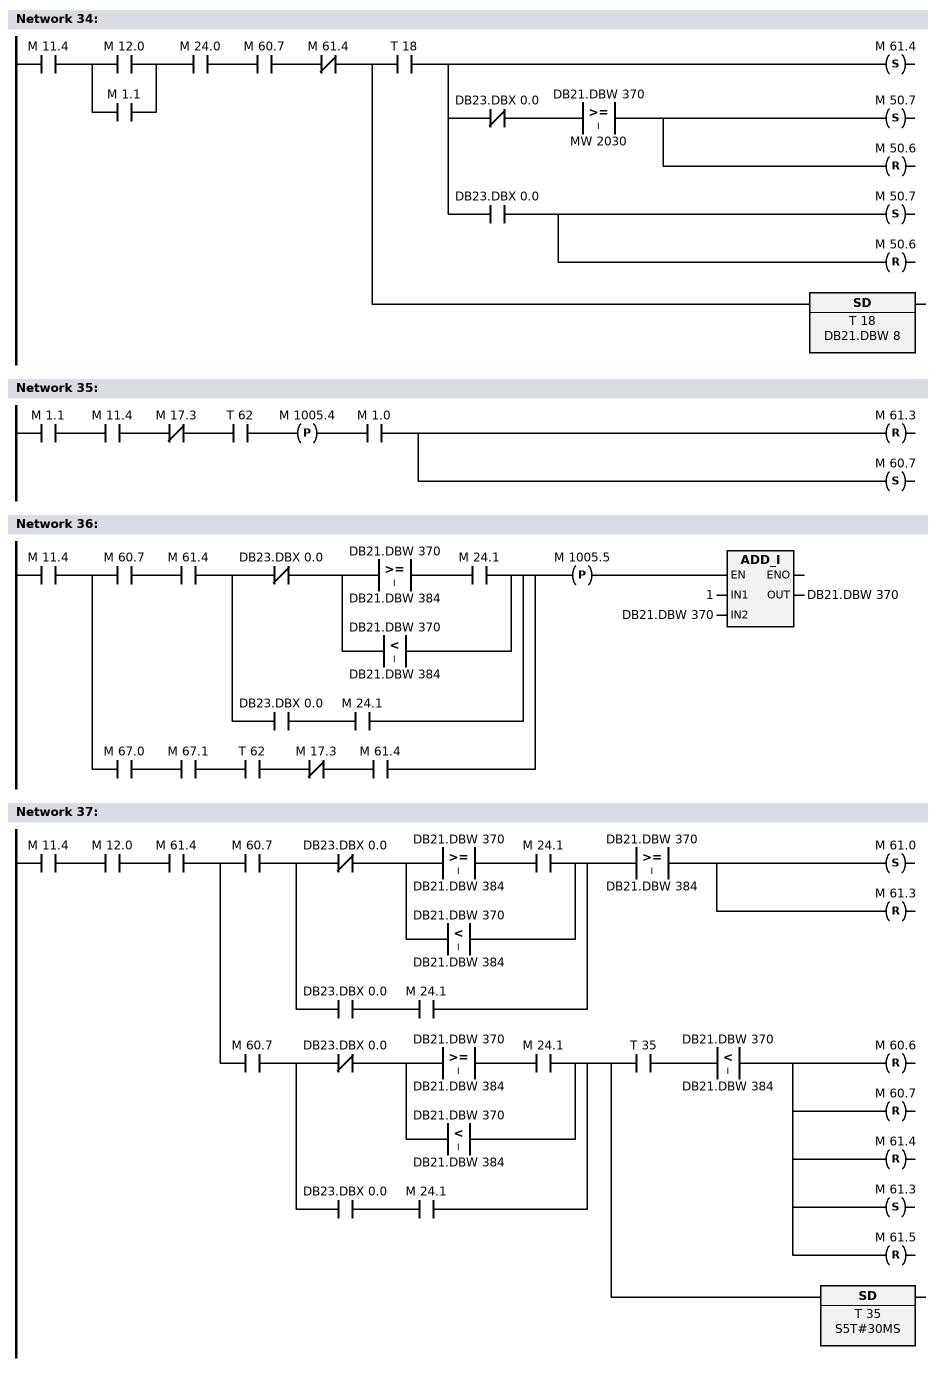
NETWORK
TITLE =
      A     M 11.4;
      A(;
      O     M 12.0;
      O     M 1.1;
      );
      A     M 24.0;
      A     M 60.7;
      AN    M 61.4;
      =     L 24.0;
      A     L 24.0;
      A     T 18;
      =     L 24.1;
      A     L 24.1;
      BLD   102;
      S     M 61.4;
      A     L 24.1;
      AN    DB23.DBX 0.0;
      A(;
      L     DB21.DBW 370;
      L     MW 2030;
      >=I;
      );
      S     M 50.7;
      R     M 50.6;
      A     L 24.1;
      A     DB23.DBX 0.0;
      S     M 50.7;
      R     M 50.6;
      A     L 24.0;
      BLD   102;
      L     DB21.DBW 8;
      SD    T 18;
NETWORK
TITLE =
      A     M 1.1;
      A     M 11.4;
      AN    M 17.3;
      A     T 62;
      FP    M 1005.4;
      A     M 1.0;
      R     M 61.3;
      S     M 60.7;
NETWORK
TITLE =
      A     M 11.4;
      A(;
      A     M 60.7;
      A     M 61.4;
      A(;
      AN    DB23.DBX 0.0;
      A(;
      A(;
      L     DB21.DBW 370;
      L     DB21.DBW 384;
      >=I;
      );
      A     M 24.1;
      O(;
      L     DB21.DBW 370;
      L     DB21.DBW 384;
      <I;
      );
      );
      O;
      A     DB23.DBX 0.0;
      A     M 24.1;
      );
      O;
      A     M 67.0;
      A     M 67.1;
      A     T 62;
      AN    M 17.3;
      A     M 61.4;
      );
      FP    M 1005.5;
      JNB   M025;
      L     1;
      L     DB21.DBW 370;
      +I;
      T     DB21.DBW 370;
M025: NOP   0;
NETWORK
TITLE =
      A     M 11.4;
      A     M 12.0;
      A     M 61.4;
      =     L 24.0;
      A     L 24.0;
      A     M 60.7;
      A(;
      AN    DB23.DBX 0.0;
      A(;
      A(;
      L     DB21.DBW 370;
      L     DB21.DBW 384;
      >=I;
      );
      A     M 24.1;
      O(;
      L     DB21.DBW 370;
      L     DB21.DBW 384;
      <I;
      );
      );
      O;
      A     DB23.DBX 0.0;
      A     M 24.1;
      );
      A(;
      L     DB21.DBW 370;
      L     DB21.DBW 384;
      >=I;
      );
      S     M 61.0;
      R     M 61.3;
      A     L 24.0;
      A     M 60.7;
      A(;
      AN    DB23.DBX 0.0;
      A(;
      A(;
      L     DB21.DBW 370;
      L     DB21.DBW 384;
      >=I;
      );
      A     M 24.1;
      O(;
      L     DB21.DBW 370;
      L     DB21.DBW 384;
      <I;
      );
      );
      O;
      A     DB23.DBX 0.0;
      A     M 24.1;
      );
      =     L 24.1;
      A     L 24.1;
      A     T 35;
      A(;
      L     DB21.DBW 370;
      L     DB21.DBW 384;
      <I;
      );
      R     M 60.6;
      R     M 60.7;
      R     M 61.4;
      S     M 61.3;
      R     M 61.5;
      A     L 24.1;
      BLD   102;
      L     S5T#30MS;
      SD    T 35;
NETWORK
TITLE =
NETWORK
TITLE =
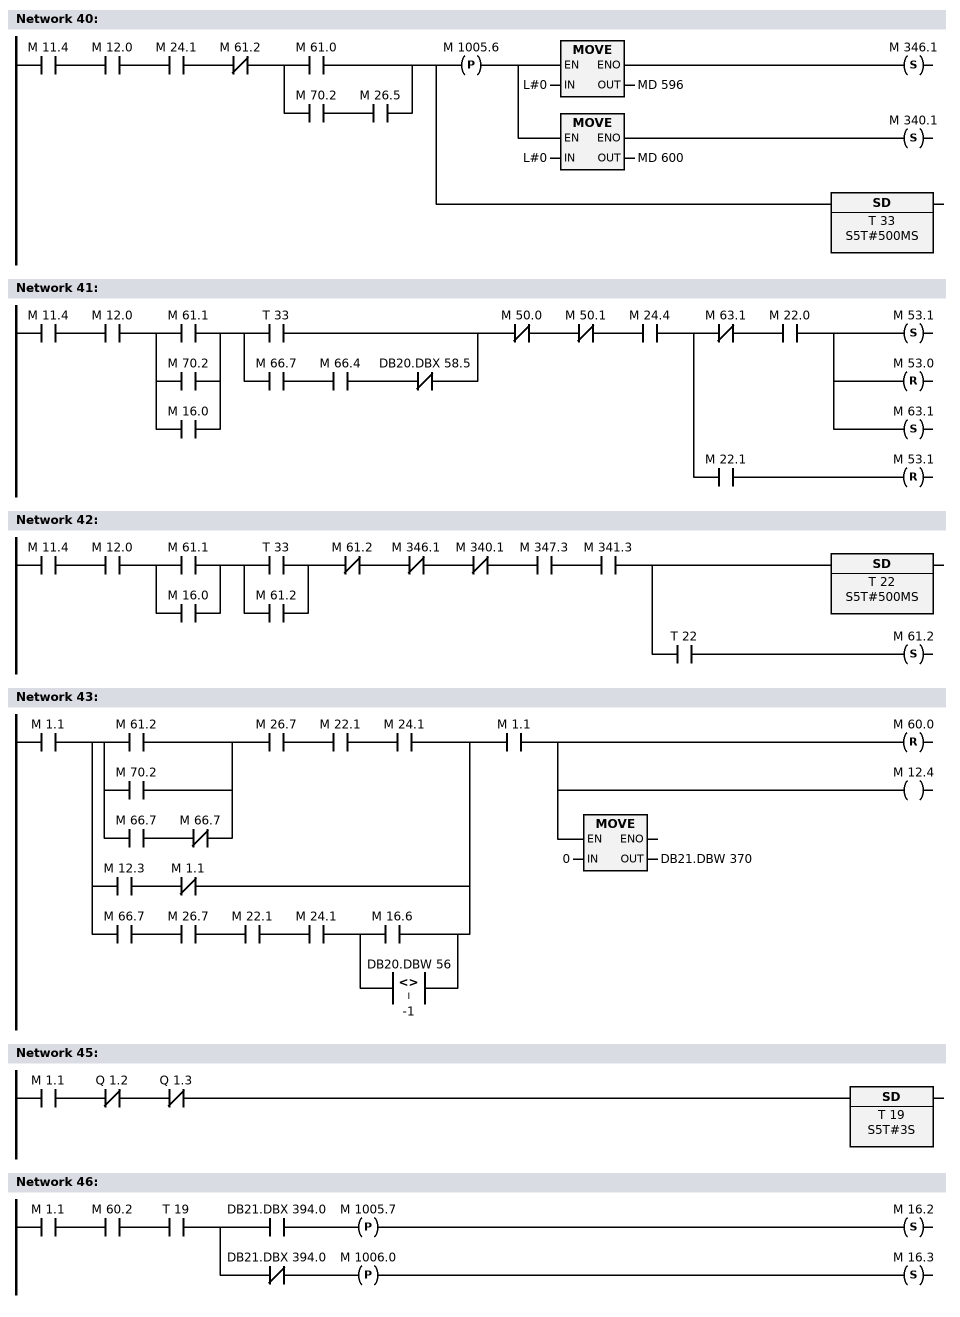
NETWORK
TITLE =
      A     M 11.4;
      A     M 12.0;
      A     M 24.1;
      AN    M 61.2;
      A(;
      O     M 61.0;
      O;
      A     M 70.2;
      A     M 26.5;
      );
      =     L 24.0;
      A     L 24.0;
      FP    M 1005.6;
      =     L 24.1;
      A     L 24.1;
      JNB   M026;
      L     L#0;
      T     MD 596;
      SET;
      SAVE;
      CLR;
M026: A     BR;
      S     M 346.1;
      A     L 24.1;
      JNB   M027;
      L     L#0;
      T     MD 600;
      SET;
      SAVE;
      CLR;
M027: A     BR;
      S     M 340.1;
      A     L 24.0;
      BLD   102;
      L     S5T#500MS;
      SD    T 33;
NETWORK
TITLE =
      A     M 11.4;
      A     M 12.0;
      A(;
      O     M 61.1;
      O     M 70.2;
      O     M 16.0;
      );
      A(;
      O     T 33;
      O;
      A     M 66.7;
      A     M 66.4;
      AN    DB20.DBX 58.5;
      );
      AN    M 50.0;
      AN    M 50.1;
      A     M 24.4;
      =     L 24.0;
      A     L 24.0;
      AN    M 63.1;
      A     M 22.0;
      S     M 53.1;
      R     M 53.0;
      S     M 63.1;
      A     L 24.0;
      A     M 22.1;
      R     M 53.1;
NETWORK
TITLE =
      A     M 11.4;
      A     M 12.0;
      A(;
      O     M 61.1;
      O     M 16.0;
      );
      A(;
      O     T 33;
      O     M 61.2;
      );
      AN    M 61.2;
      AN    M 346.1;
      AN    M 340.1;
      A     M 347.3;
      A     M 341.3;
      =     L 24.0;
      A     L 24.0;
      BLD   102;
      L     S5T#500MS;
      SD    T 22;
      A     L 24.0;
      A     T 22;
      S     M 61.2;
NETWORK
TITLE =
      A     M 1.1;
      A(;
      A(;
      O     M 61.2;
      O     M 70.2;
      O;
      A     M 66.7;
      AN    M 66.7;
      );
      A     M 26.7;
      A     M 22.1;
      A     M 24.1;
      O;
      A     M 12.3;
      AN    M 1.1;
      O;
      A     M 66.7;
      A     M 26.7;
      A     M 22.1;
      A     M 24.1;
      A(;
      O     M 16.6;
      O(;
      L     DB20.DBW 56;
      L     -1;
      <>I;
      );
      );
      );
      A     M 1.1;
      =     L 24.0;
      A     L 24.0;
      BLD   102;
      R     M 60.0;
      A     L 24.0;
      BLD   102;
      =     M 12.4;
      A     L 24.0;
      JNB   M028;
      L     0;
      T     DB21.DBW 370;
M028: NOP   0;
NETWORK
TITLE =
NETWORK
TITLE =
      A     M 1.1;
      AN    Q 1.2;
      AN    Q 1.3;
      L     S5T#3S;
      SD    T 19;
NETWORK
TITLE =
      A     M 1.1;
      A     M 60.2;
      A     T 19;
      =     L 24.0;
      A     L 24.0;
      A     DB21.DBX 394.0;
      FP    M 1005.7;
      S     M 16.2;
      A     L 24.0;
      AN    DB21.DBX 394.0;
      FP    M 1006.0;
      S     M 16.3;
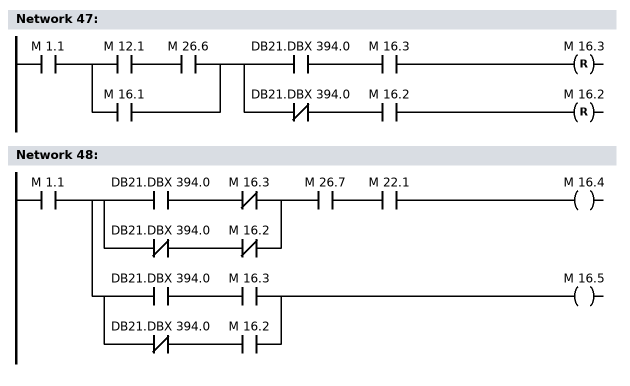
NETWORK
TITLE =
      A     M 1.1;
      A(;
      A     M 12.1;
      A     M 26.6;
      O     M 16.1;
      );
      =     L 24.0;
      A     L 24.0;
      A     DB21.DBX 394.0;
      A     M 16.3;
      R     M 16.3;
      A     L 24.0;
      AN    DB21.DBX 394.0;
      A     M 16.2;
      R     M 16.2;
NETWORK
TITLE =
      A     M 1.1;
      =     L 24.0;
      A     L 24.0;
      A(;
      A     DB21.DBX 394.0;
      AN    M 16.3;
      O;
      AN    DB21.DBX 394.0;
      AN    M 16.2;
      );
      A     M 26.7;
      A     M 22.1;
      =     M 16.4;
      A     L 24.0;
      A(;
      A     DB21.DBX 394.0;
      A     M 16.3;
      O;
      AN    DB21.DBX 394.0;
      A     M 16.2;
      );
      =     M 16.5;
END_FUNCTION

FUNCTION FC 16 : VOID
VERSION : 0.1
BEGIN
// (block stored without names or comments; labels and parameter names are numbered)
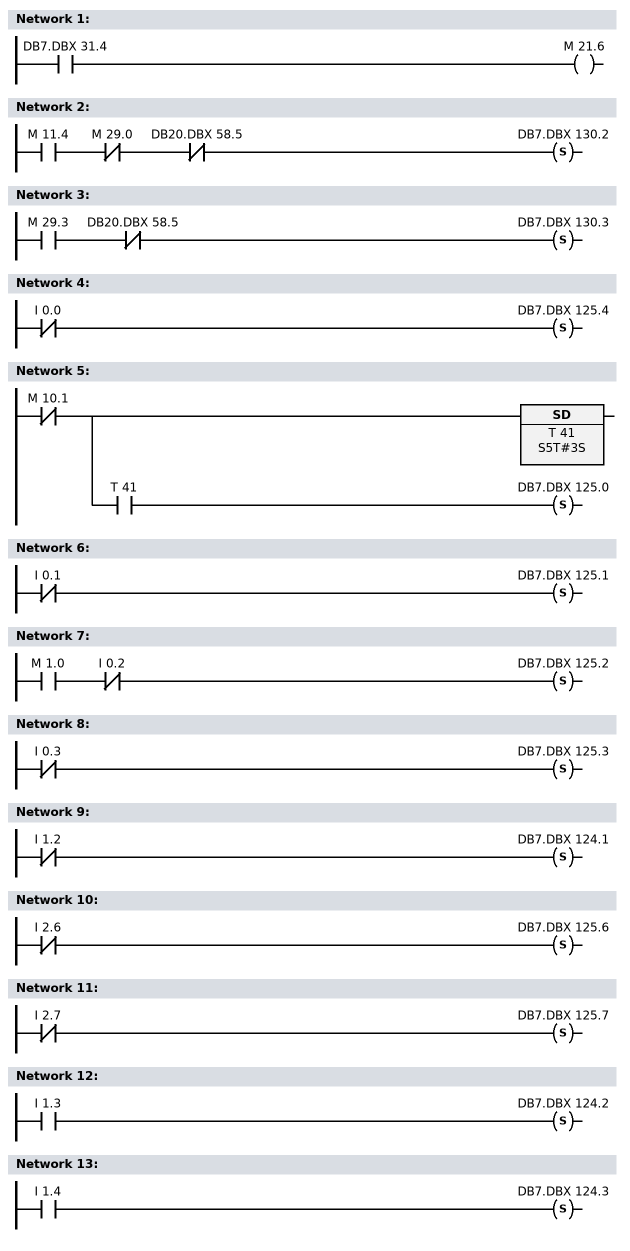
NETWORK
TITLE =
      A     DB7.DBX 31.4;
      =     M 21.6;
NETWORK
TITLE =
      A     M 11.4;
      AN    M 29.0;
      AN    DB20.DBX 58.5;
      S     DB7.DBX 130.2;
NETWORK
TITLE =
      A     M 29.3;
      AN    DB20.DBX 58.5;
      S     DB7.DBX 130.3;
NETWORK
TITLE =
      AN    I 0.0;
      S     DB7.DBX 125.4;
NETWORK
TITLE =
      AN    M 10.1;
      =     L 1.0;
      A     L 1.0;
      BLD   102;
      L     S5T#3S;
      SD    T 41;
      A     L 1.0;
      A     T 41;
      S     DB7.DBX 125.0;
NETWORK
TITLE =
      AN    I 0.1;
      S     DB7.DBX 125.1;
NETWORK
TITLE =
      A     M 1.0;
      AN    I 0.2;
      S     DB7.DBX 125.2;
NETWORK
TITLE =
      AN    I 0.3;
      S     DB7.DBX 125.3;
NETWORK
TITLE =
      AN    I 1.2;
      S     DB7.DBX 124.1;
NETWORK
TITLE =
      AN    I 2.6;
      S     DB7.DBX 125.6;
NETWORK
TITLE =
      AN    I 2.7;
      S     DB7.DBX 125.7;
NETWORK
TITLE =
      A     I 1.3;
      S     DB7.DBX 124.2;
NETWORK
TITLE =
      A     I 1.4;
      S     DB7.DBX 124.3;
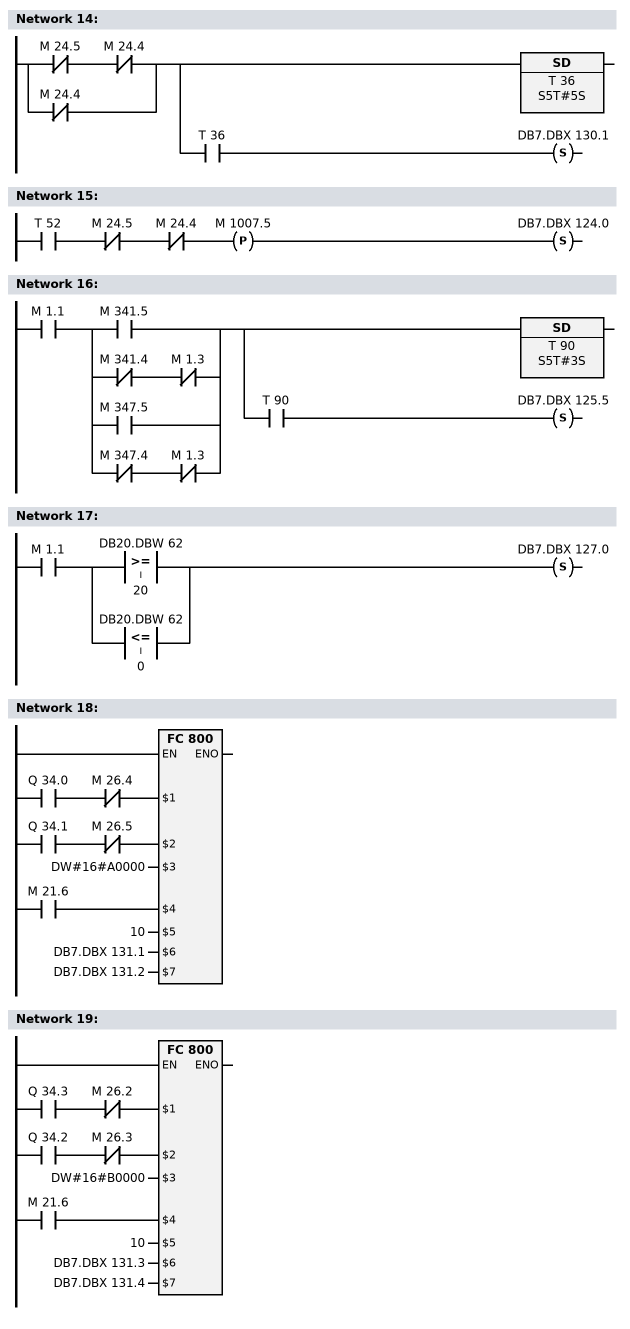
NETWORK
TITLE =
      AN    M 24.5;
      AN    M 24.4;
      ON    M 24.4;
      =     L 1.0;
      A     L 1.0;
      BLD   102;
      L     S5T#5S;
      SD    T 36;
      A     L 1.0;
      A     T 36;
      S     DB7.DBX 130.1;
NETWORK
TITLE =
      A     T 52;
      AN    M 24.5;
      AN    M 24.4;
      FP    M 1007.5;
      S     DB7.DBX 124.0;
NETWORK
TITLE =
      A     M 1.1;
      A(;
      O     M 341.5;
      O;
      AN    M 341.4;
      AN    M 1.3;
      O     M 347.5;
      O;
      AN    M 347.4;
      AN    M 1.3;
      );
      =     L 1.0;
      A     L 1.0;
      BLD   102;
      L     S5T#3S;
      SD    T 90;
      A     L 1.0;
      A     T 90;
      S     DB7.DBX 125.5;
NETWORK
TITLE =
      A     M 1.1;
      A(;
      O(;
      L     DB20.DBW 62;
      L     20;
      >=I;
      );
      O(;
      L     DB20.DBW 62;
      L     0;
      <=I;
      );
      );
      S     DB7.DBX 127.0;
NETWORK
TITLE =
      A     Q 34.0;
      AN    M 26.4;
      =     L 1.0;
      BLD   103;
      A     Q 34.1;
      AN    M 26.5;
      =     L 1.1;
      BLD   103;
      A     M 21.6;
      =     L 1.2;
      BLD   103;
      CALL  FC 800 (
           $1                       := L 1.0,
           $2                       := L 1.1,
           $3                       := DW#16#A0000,
           $4                       := L 1.2,
           $5                       := 10,
           $6                       := DB7.DBX 131.1,
           $7                       := DB7.DBX 131.2);
      NOP   0;
NETWORK
TITLE =
      A     Q 34.3;
      AN    M 26.2;
      =     L 1.0;
      BLD   103;
      A     Q 34.2;
      AN    M 26.3;
      =     L 1.1;
      BLD   103;
      A     M 21.6;
      =     L 1.2;
      BLD   103;
      CALL  FC 800 (
           $1                       := L 1.0,
           $2                       := L 1.1,
           $3                       := DW#16#B0000,
           $4                       := L 1.2,
           $5                       := 10,
           $6                       := DB7.DBX 131.3,
           $7                       := DB7.DBX 131.4);
      NOP   0;
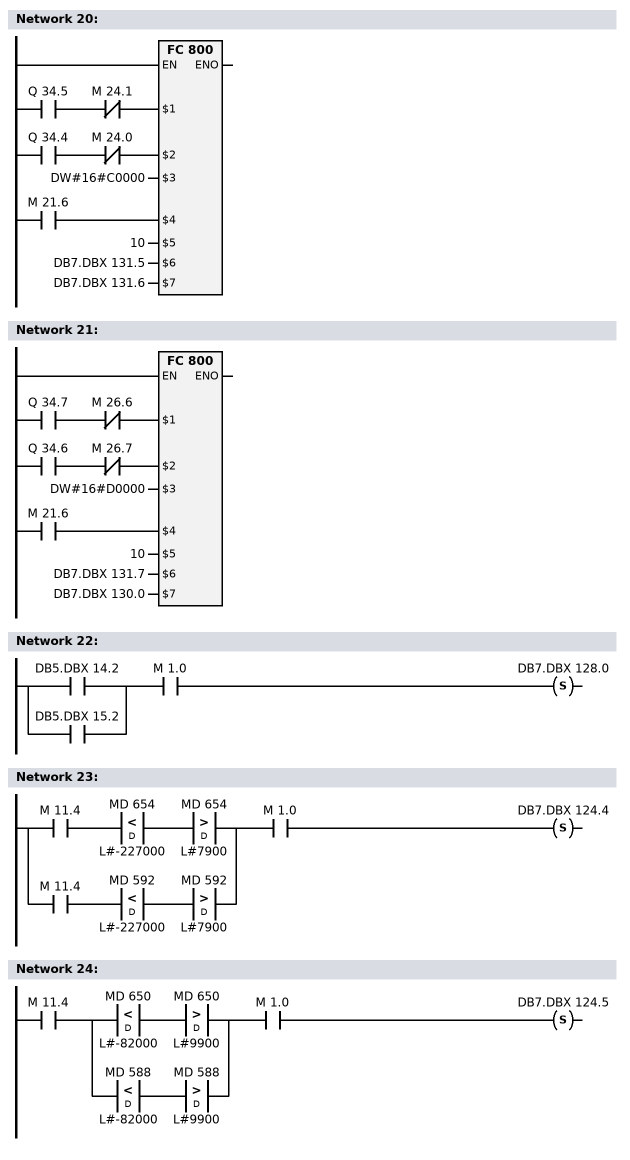
NETWORK
TITLE =
      A     Q 34.5;
      AN    M 24.1;
      =     L 1.0;
      BLD   103;
      A     Q 34.4;
      AN    M 24.0;
      =     L 1.1;
      BLD   103;
      A     M 21.6;
      =     L 1.2;
      BLD   103;
      CALL  FC 800 (
           $1                       := L 1.0,
           $2                       := L 1.1,
           $3                       := DW#16#C0000,
           $4                       := L 1.2,
           $5                       := 10,
           $6                       := DB7.DBX 131.5,
           $7                       := DB7.DBX 131.6);
      NOP   0;
NETWORK
TITLE =
      A     Q 34.7;
      AN    M 26.6;
      =     L 1.0;
      BLD   103;
      A     Q 34.6;
      AN    M 26.7;
      =     L 1.1;
      BLD   103;
      A     M 21.6;
      =     L 1.2;
      BLD   103;
      CALL  FC 800 (
           $1                       := L 1.0,
           $2                       := L 1.1,
           $3                       := DW#16#D0000,
           $4                       := L 1.2,
           $5                       := 10,
           $6                       := DB7.DBX 131.7,
           $7                       := DB7.DBX 130.0);
      NOP   0;
NETWORK
TITLE =
      A(;
      O     DB5.DBX 14.2;
      O     DB5.DBX 15.2;
      );
      A     M 1.0;
      S     DB7.DBX 128.0;
NETWORK
TITLE =
      A(;
      A     M 11.4;
      A(;
      L     MD 654;
      L     L#-227000;
      <D;
      );
      A(;
      L     MD 654;
      L     L#7900;
      >D;
      );
      O;
      A     M 11.4;
      A(;
      L     MD 592;
      L     L#-227000;
      <D;
      );
      A(;
      L     MD 592;
      L     L#7900;
      >D;
      );
      );
      A     M 1.0;
      S     DB7.DBX 124.4;
NETWORK
TITLE =
      A     M 11.4;
      A(;
      A(;
      L     MD 650;
      L     L#-82000;
      <D;
      );
      A(;
      L     MD 650;
      L     L#9900;
      >D;
      );
      O;
      A(;
      L     MD 588;
      L     L#-82000;
      <D;
      );
      A(;
      L     MD 588;
      L     L#9900;
      >D;
      );
      );
      A     M 1.0;
      S     DB7.DBX 124.5;
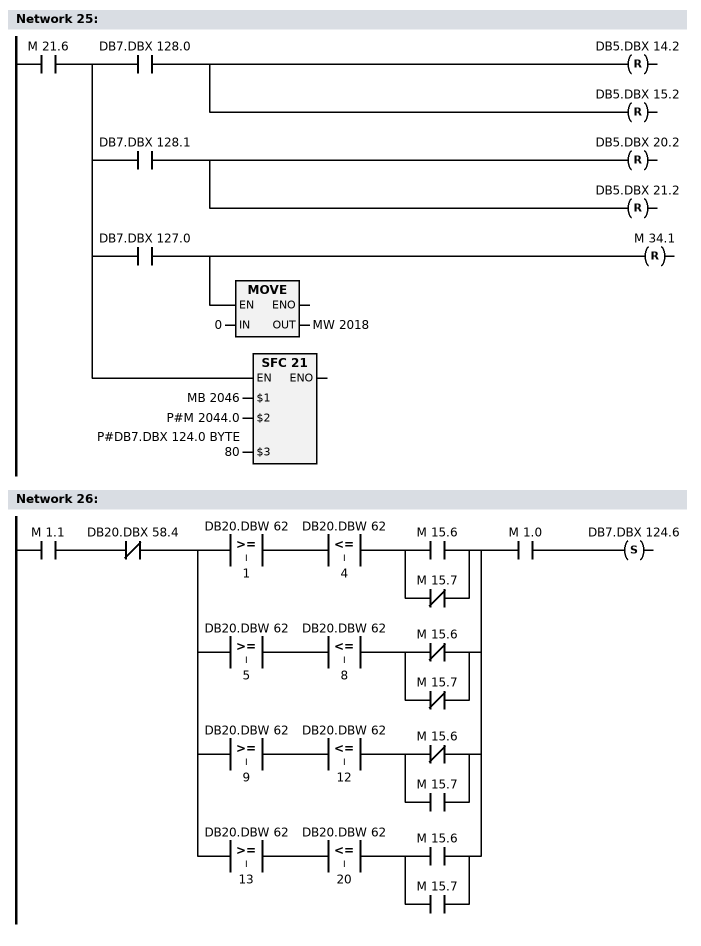
NETWORK
TITLE =
      A     M 21.6;
      =     L 1.0;
      A     L 1.0;
      A     DB7.DBX 128.0;
      R     DB5.DBX 14.2;
      R     DB5.DBX 15.2;
      A     L 1.0;
      A     DB7.DBX 128.1;
      R     DB5.DBX 20.2;
      R     DB5.DBX 21.2;
      A     L 1.0;
      A     DB7.DBX 127.0;
      =     L 1.1;
      A     L 1.1;
      BLD   102;
      R     M 34.1;
      A     L 1.1;
      JNB   M001;
      L     0;
      T     MW 2018;
M001: NOP   0;
      A     L 1.0;
      JNB   M002;
      CALL  SFC 21 (
           $1                       := MB 2046,
           $2                       := P#M 2044.0,
           $3                       := P#DB7.DBX 124.0 BYTE 80);
M002: NOP   0;
NETWORK
TITLE =
      A     M 1.1;
      AN    DB20.DBX 58.4;
      A(;
      A(;
      L     DB20.DBW 62;
      L     1;
      >=I;
      );
      A(;
      L     DB20.DBW 62;
      L     4;
      <=I;
      );
      A(;
      O     M 15.6;
      ON    M 15.7;
      );
      O;
      A(;
      L     DB20.DBW 62;
      L     5;
      >=I;
      );
      A(;
      L     DB20.DBW 62;
      L     8;
      <=I;
      );
      A(;
      ON    M 15.6;
      ON    M 15.7;
      );
      O;
      A(;
      L     DB20.DBW 62;
      L     9;
      >=I;
      );
      A(;
      L     DB20.DBW 62;
      L     12;
      <=I;
      );
      A(;
      ON    M 15.6;
      O     M 15.7;
      );
      O;
      A(;
      L     DB20.DBW 62;
      L     13;
      >=I;
      );
      A(;
      L     DB20.DBW 62;
      L     20;
      <=I;
      );
      A(;
      O     M 15.6;
      O     M 15.7;
      );
      );
      A     M 1.0;
      S     DB7.DBX 124.6;
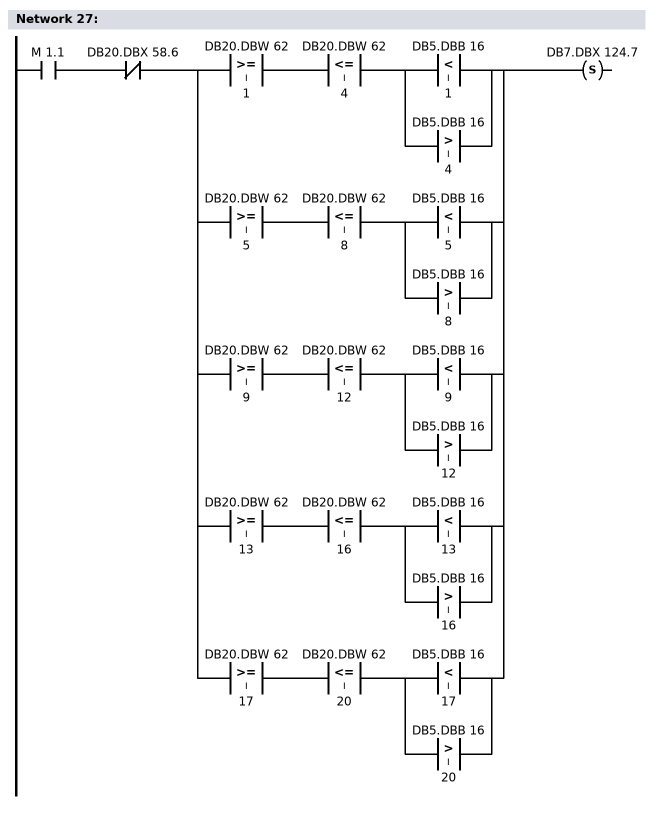
NETWORK
TITLE =
      A     M 1.1;
      AN    DB20.DBX 58.6;
      A(;
      A(;
      L     DB20.DBW 62;
      L     1;
      >=I;
      );
      A(;
      L     DB20.DBW 62;
      L     4;
      <=I;
      );
      A(;
      O(;
      L     DB5.DBB 16;
      L     1;
      <I;
      );
      O(;
      L     DB5.DBB 16;
      L     4;
      >I;
      );
      );
      O;
      A(;
      L     DB20.DBW 62;
      L     5;
      >=I;
      );
      A(;
      L     DB20.DBW 62;
      L     8;
      <=I;
      );
      A(;
      O(;
      L     DB5.DBB 16;
      L     5;
      <I;
      );
      O(;
      L     DB5.DBB 16;
      L     8;
      >I;
      );
      );
      O;
      A(;
      L     DB20.DBW 62;
      L     9;
      >=I;
      );
      A(;
      L     DB20.DBW 62;
      L     12;
      <=I;
      );
      A(;
      O(;
      L     DB5.DBB 16;
      L     9;
      <I;
      );
      O(;
      L     DB5.DBB 16;
      L     12;
      >I;
      );
      );
      O;
      A(;
      L     DB20.DBW 62;
      L     13;
      >=I;
      );
      A(;
      L     DB20.DBW 62;
      L     16;
      <=I;
      );
      A(;
      O(;
      L     DB5.DBB 16;
      L     13;
      <I;
      );
      O(;
      L     DB5.DBB 16;
      L     16;
      >I;
      );
      );
      O;
      A(;
      L     DB20.DBW 62;
      L     17;
      >=I;
      );
      A(;
      L     DB20.DBW 62;
      L     20;
      <=I;
      );
      A(;
      O(;
      L     DB5.DBB 16;
      L     17;
      <I;
      );
      O(;
      L     DB5.DBB 16;
      L     20;
      >I;
      );
      );
      );
      S     DB7.DBX 124.7;
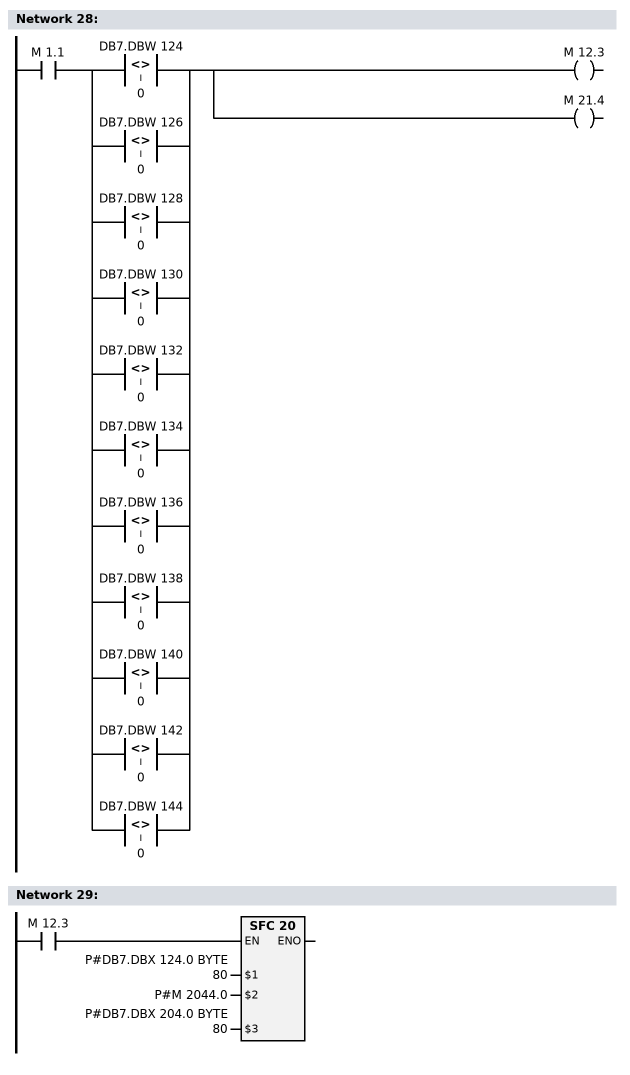
NETWORK
TITLE =
      A     M 1.1;
      A(;
      O(;
      L     DB7.DBW 124;
      L     0;
      <>I;
      );
      O(;
      L     DB7.DBW 126;
      L     0;
      <>I;
      );
      O(;
      L     DB7.DBW 128;
      L     0;
      <>I;
      );
      O(;
      L     DB7.DBW 130;
      L     0;
      <>I;
      );
      O(;
      L     DB7.DBW 132;
      L     0;
      <>I;
      );
      O(;
      L     DB7.DBW 134;
      L     0;
      <>I;
      );
      O(;
      L     DB7.DBW 136;
      L     0;
      <>I;
      );
      O(;
      L     DB7.DBW 138;
      L     0;
      <>I;
      );
      O(;
      L     DB7.DBW 140;
      L     0;
      <>I;
      );
      O(;
      L     DB7.DBW 142;
      L     0;
      <>I;
      );
      O(;
      L     DB7.DBW 144;
      L     0;
      <>I;
      );
      );
      =     M 12.3;
      =     M 21.4;
NETWORK
TITLE =
      A     M 12.3;
      JNB   M003;
      CALL  SFC 20 (
           $1                       := P#DB7.DBX 124.0 BYTE 80,
           $2                       := P#M 2044.0,
           $3                       := P#DB7.DBX 204.0 BYTE 80);
M003: NOP   0;
END_FUNCTION

FUNCTION FC 17 : VOID
VERSION : 0.1
BEGIN
// (block stored without names or comments; labels and parameter names are numbered)
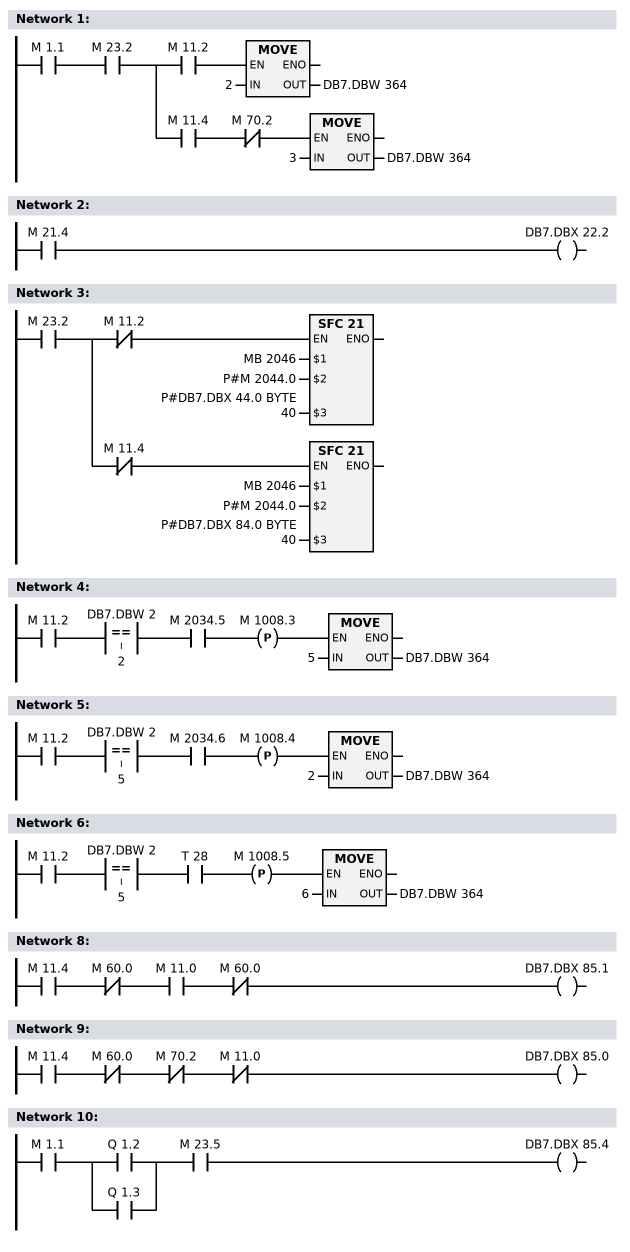
NETWORK
TITLE =
      A     M 1.1;
      A     M 23.2;
      =     L 0.0;
      A     L 0.0;
      A     M 11.2;
      JNB   M001;
      L     2;
      T     DB7.DBW 364;
M001: NOP   0;
      A     L 0.0;
      A     M 11.4;
      AN    M 70.2;
      JNB   M002;
      L     3;
      T     DB7.DBW 364;
M002: NOP   0;
NETWORK
TITLE =
      A     M 21.4;
      =     DB7.DBX 22.2;
NETWORK
TITLE =
      A     M 23.2;
      =     L 0.0;
      A     L 0.0;
      AN    M 11.2;
      JNB   M003;
      CALL  SFC 21 (
           $1                       := MB 2046,
           $2                       := P#M 2044.0,
           $3                       := P#DB7.DBX 44.0 BYTE 40);
M003: NOP   0;
      A     L 0.0;
      AN    M 11.4;
      JNB   M004;
      CALL  SFC 21 (
           $1                       := MB 2046,
           $2                       := P#M 2044.0,
           $3                       := P#DB7.DBX 84.0 BYTE 40);
M004: NOP   0;
NETWORK
TITLE =
      A     M 11.2;
      A(;
      L     DB7.DBW 2;
      L     2;
      ==I;
      );
      A     M 2034.5;
      FP    M 1008.3;
      JNB   M005;
      L     5;
      T     DB7.DBW 364;
M005: NOP   0;
NETWORK
TITLE =
      A     M 11.2;
      A(;
      L     DB7.DBW 2;
      L     5;
      ==I;
      );
      A     M 2034.6;
      FP    M 1008.4;
      JNB   M006;
      L     2;
      T     DB7.DBW 364;
M006: NOP   0;
NETWORK
TITLE =
      A     M 11.2;
      A(;
      L     DB7.DBW 2;
      L     5;
      ==I;
      );
      A     T 28;
      FP    M 1008.5;
      JNB   M007;
      L     6;
      T     DB7.DBW 364;
M007: NOP   0;
NETWORK
TITLE =
NETWORK
TITLE =
      A     M 11.4;
      AN    M 60.0;
      A     M 11.0;
      AN    M 60.0;
      =     DB7.DBX 85.1;
NETWORK
TITLE =
      A     M 11.4;
      AN    M 60.0;
      AN    M 70.2;
      AN    M 11.0;
      =     DB7.DBX 85.0;
NETWORK
TITLE =
      A     M 1.1;
      A(;
      O     Q 1.2;
      O     Q 1.3;
      );
      A     M 23.5;
      =     DB7.DBX 85.4;
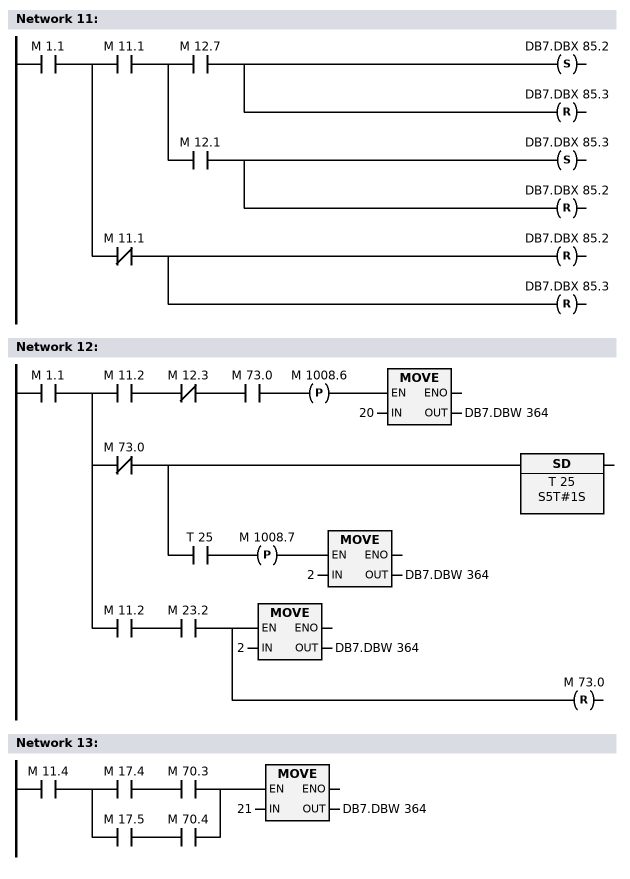
NETWORK
TITLE =
      A     M 1.1;
      =     L 0.0;
      A     L 0.0;
      A     M 11.1;
      =     L 0.1;
      A     L 0.1;
      A     M 12.7;
      S     DB7.DBX 85.2;
      R     DB7.DBX 85.3;
      A     L 0.1;
      A     M 12.1;
      S     DB7.DBX 85.3;
      R     DB7.DBX 85.2;
      A     L 0.0;
      AN    M 11.1;
      R     DB7.DBX 85.2;
      R     DB7.DBX 85.3;
NETWORK
TITLE =
      A     M 1.1;
      =     L 0.0;
      A     L 0.0;
      A     M 11.2;
      AN    M 12.3;
      A     M 73.0;
      FP    M 1008.6;
      JNB   M008;
      L     20;
      T     DB7.DBW 364;
M008: NOP   0;
      A     L 0.0;
      AN    M 73.0;
      =     L 0.1;
      A     L 0.1;
      BLD   102;
      L     S5T#1S;
      SD    T 25;
      A     L 0.1;
      A     T 25;
      FP    M 1008.7;
      JNB   M009;
      L     2;
      T     DB7.DBW 364;
M009: NOP   0;
      A     L 0.0;
      A     M 11.2;
      A     M 23.2;
      =     L 0.1;
      A     L 0.1;
      JNB   M010;
      L     2;
      T     DB7.DBW 364;
M010: NOP   0;
      A     L 0.1;
      BLD   102;
      R     M 73.0;
NETWORK
TITLE =
      A     M 11.4;
      A(;
      A     M 17.4;
      A     M 70.3;
      O;
      A     M 17.5;
      A     M 70.4;
      );
      JNB   M011;
      L     21;
      T     DB7.DBW 364;
M011: NOP   0;
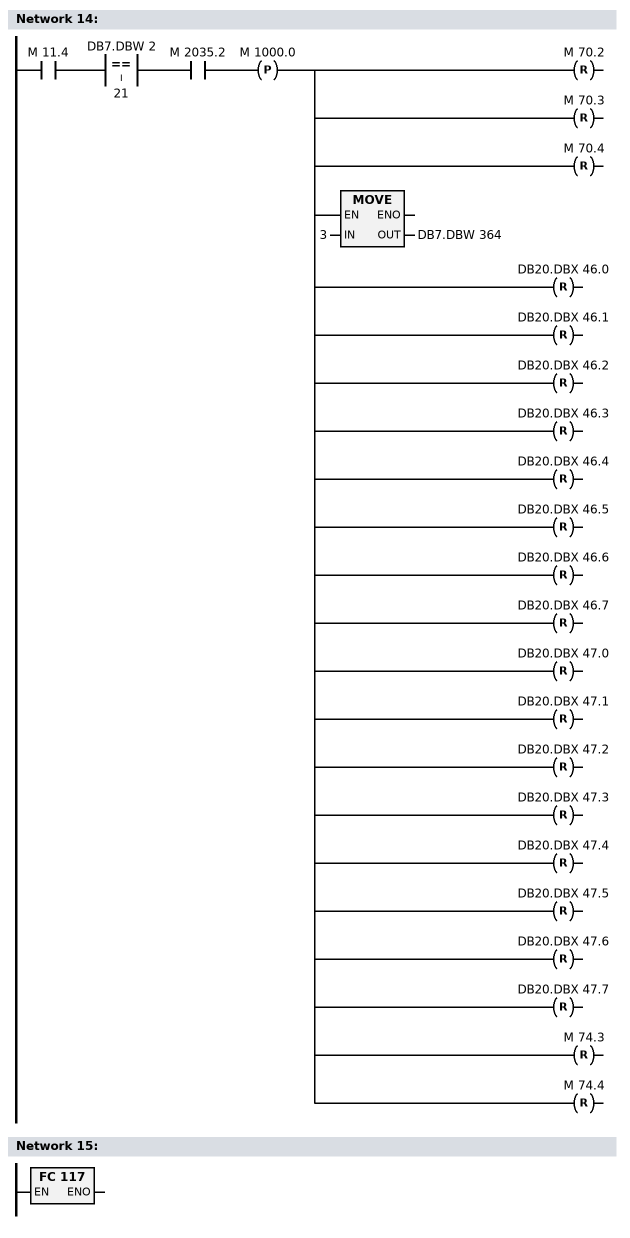
NETWORK
TITLE =
      A     M 11.4;
      A(;
      L     DB7.DBW 2;
      L     21;
      ==I;
      );
      A     M 2035.2;
      FP    M 1000.0;
      =     L 0.0;
      A     L 0.0;
      BLD   102;
      R     M 70.2;
      A     L 0.0;
      BLD   102;
      R     M 70.3;
      A     L 0.0;
      BLD   102;
      R     M 70.4;
      A     L 0.0;
      JNB   M012;
      L     3;
      T     DB7.DBW 364;
M012: NOP   0;
      A     L 0.0;
      BLD   102;
      R     DB20.DBX 46.0;
      A     L 0.0;
      BLD   102;
      R     DB20.DBX 46.1;
      A     L 0.0;
      BLD   102;
      R     DB20.DBX 46.2;
      A     L 0.0;
      BLD   102;
      R     DB20.DBX 46.3;
      A     L 0.0;
      BLD   102;
      R     DB20.DBX 46.4;
      A     L 0.0;
      BLD   102;
      R     DB20.DBX 46.5;
      A     L 0.0;
      BLD   102;
      R     DB20.DBX 46.6;
      A     L 0.0;
      BLD   102;
      R     DB20.DBX 46.7;
      A     L 0.0;
      BLD   102;
      R     DB20.DBX 47.0;
      A     L 0.0;
      BLD   102;
      R     DB20.DBX 47.1;
      A     L 0.0;
      BLD   102;
      R     DB20.DBX 47.2;
      A     L 0.0;
      BLD   102;
      R     DB20.DBX 47.3;
      A     L 0.0;
      BLD   102;
      R     DB20.DBX 47.4;
      A     L 0.0;
      BLD   102;
      R     DB20.DBX 47.5;
      A     L 0.0;
      BLD   102;
      R     DB20.DBX 47.6;
      A     L 0.0;
      BLD   102;
      R     DB20.DBX 47.7;
      A     L 0.0;
      BLD   102;
      R     M 74.3;
      A     L 0.0;
      BLD   102;
      R     M 74.4;
NETWORK
TITLE =
      CALL  FC 117;
      NOP   0;
END_FUNCTION

FUNCTION FC 18 : VOID
VERSION : 0.1
BEGIN
// (block stored without names or comments; labels and parameter names are numbered)
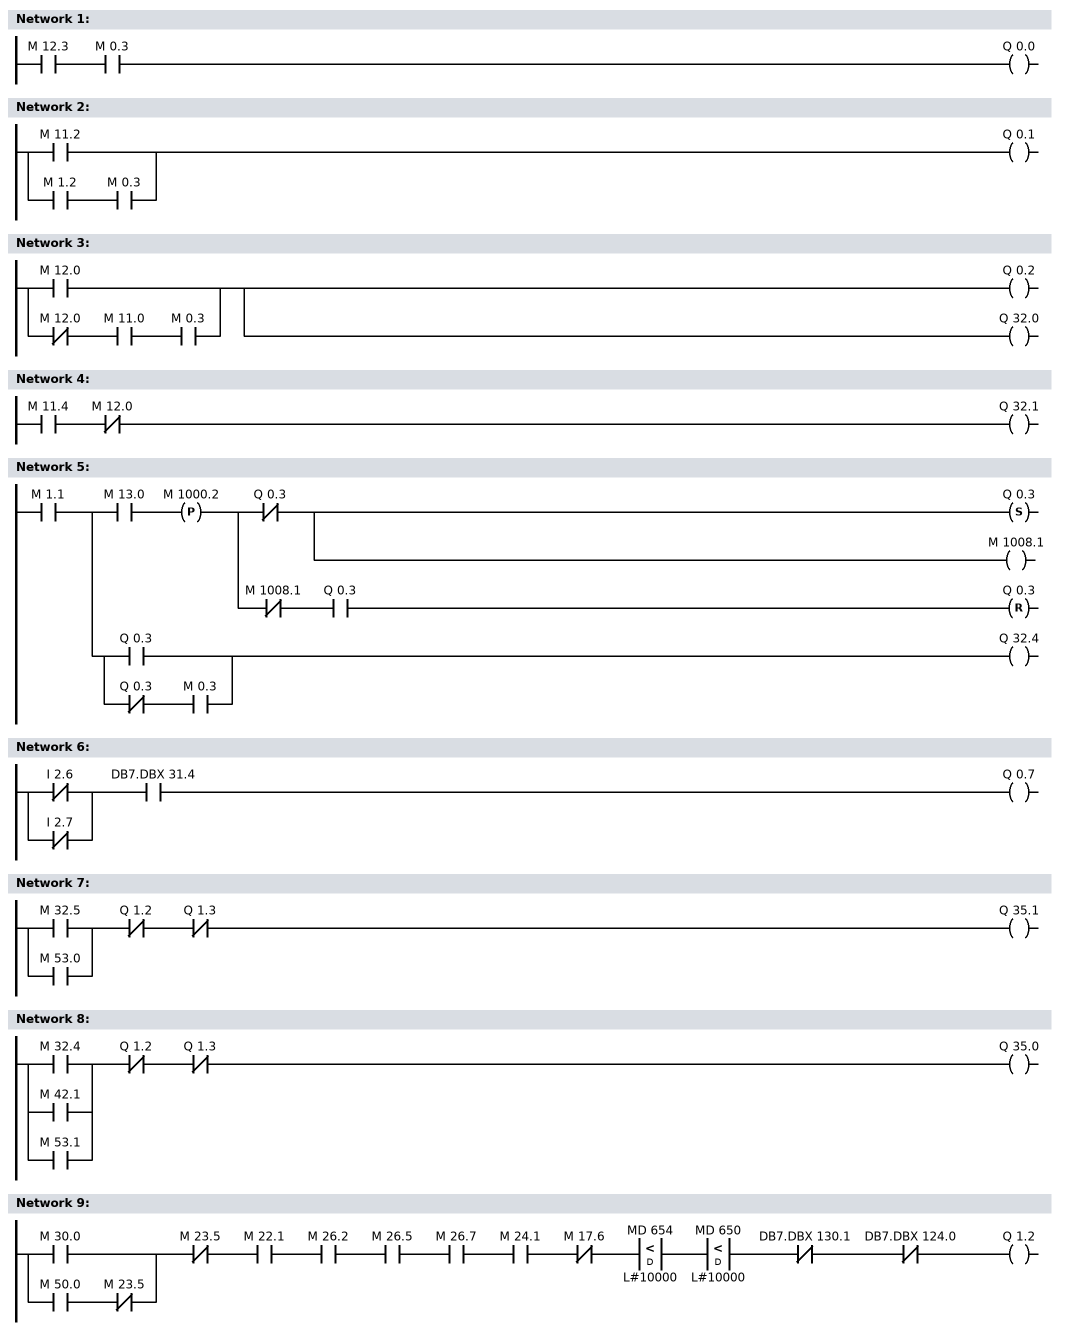
NETWORK
TITLE =
      A     M 12.3;
      A     M 0.3;
      =     Q 0.0;
NETWORK
TITLE =
      O     M 11.2;
      O;
      A     M 1.2;
      A     M 0.3;
      =     Q 0.1;
NETWORK
TITLE =
      O     M 12.0;
      O;
      AN    M 12.0;
      A     M 11.0;
      A     M 0.3;
      =     Q 0.2;
      =     Q 32.0;
NETWORK
TITLE =
      A     M 11.4;
      AN    M 12.0;
      =     Q 32.1;
NETWORK
TITLE =
      A     M 1.1;
      =     L 0.0;
      A     L 0.0;
      A     M 13.0;
      FP    M 1000.2;
      =     L 0.1;
      A     L 0.1;
      AN    Q 0.3;
      S     Q 0.3;
      =     M 1008.1;
      A     L 0.1;
      AN    M 1008.1;
      A     Q 0.3;
      R     Q 0.3;
      A     L 0.0;
      A(;
      O     Q 0.3;
      O;
      AN    Q 0.3;
      A     M 0.3;
      );
      =     Q 32.4;
NETWORK
TITLE =
      A(;
      ON    I 2.6;
      ON    I 2.7;
      );
      A     DB7.DBX 31.4;
      =     Q 0.7;
NETWORK
TITLE =
      A(;
      O     M 32.5;
      O     M 53.0;
      );
      AN    Q 1.2;
      AN    Q 1.3;
      =     Q 35.1;
NETWORK
TITLE =
      A(;
      O     M 32.4;
      O     M 42.1;
      O     M 53.1;
      );
      AN    Q 1.2;
      AN    Q 1.3;
      =     Q 35.0;
NETWORK
TITLE =
      A(;
      O     M 30.0;
      O;
      A     M 50.0;
      AN    M 23.5;
      );
      AN    M 23.5;
      A     M 22.1;
      A     M 26.2;
      A     M 26.5;
      A     M 26.7;
      A     M 24.1;
      AN    M 17.6;
      A(;
      L     MD 654;
      L     L#10000;
      <D;
      );
      A(;
      L     MD 650;
      L     L#10000;
      <D;
      );
      AN    DB7.DBX 130.1;
      AN    DB7.DBX 124.0;
      =     Q 1.2;
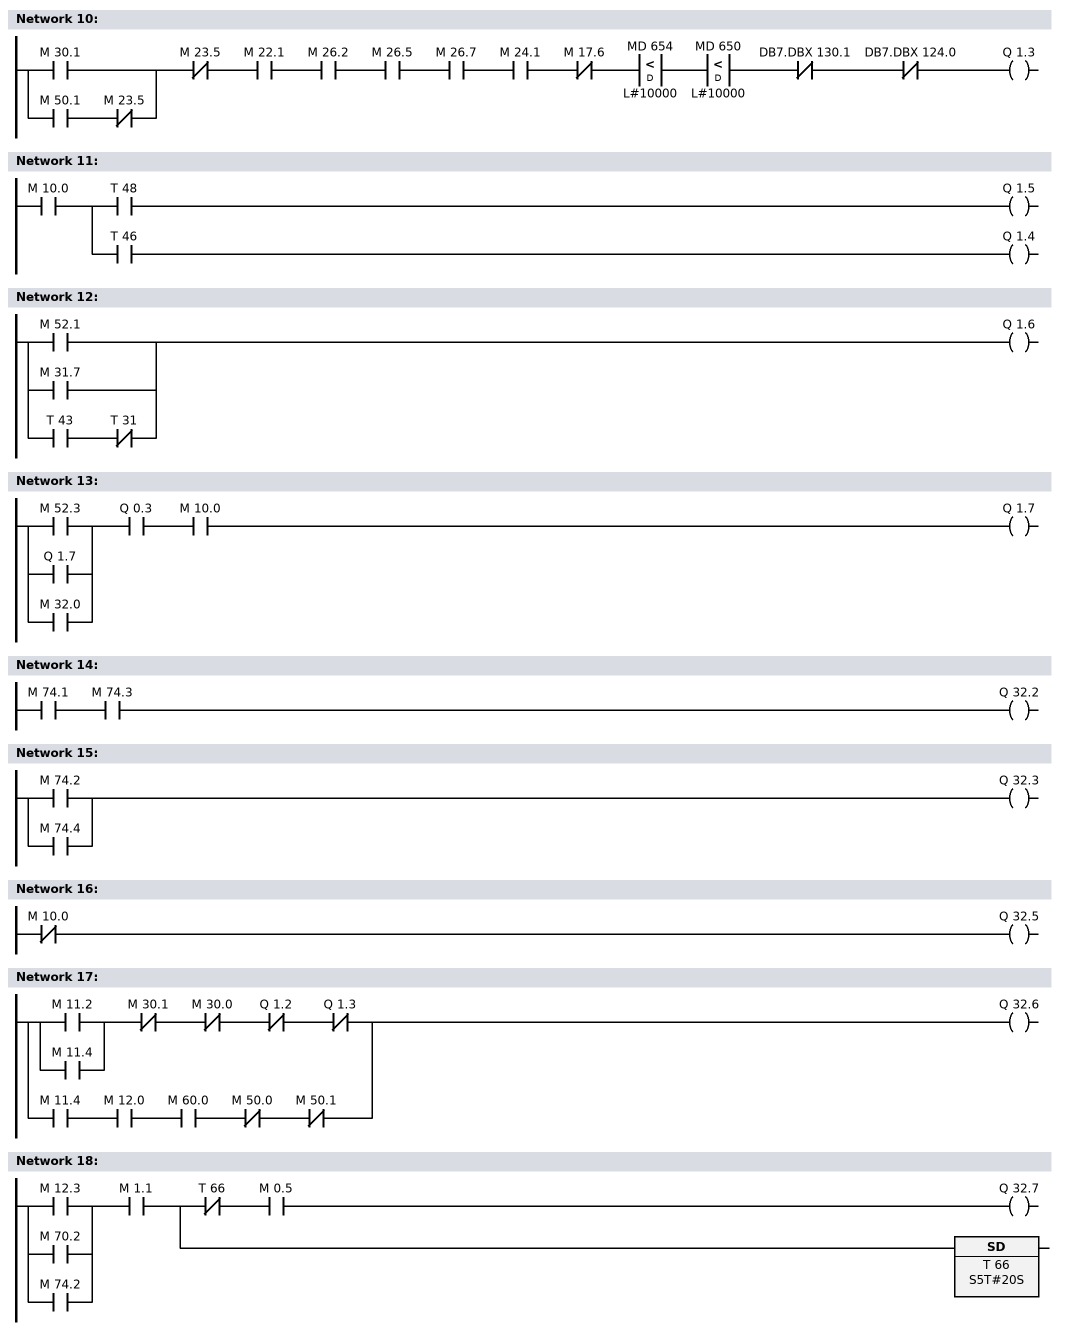
NETWORK
TITLE =
      A(;
      O     M 30.1;
      O;
      A     M 50.1;
      AN    M 23.5;
      );
      AN    M 23.5;
      A     M 22.1;
      A     M 26.2;
      A     M 26.5;
      A     M 26.7;
      A     M 24.1;
      AN    M 17.6;
      A(;
      L     MD 654;
      L     L#10000;
      <D;
      );
      A(;
      L     MD 650;
      L     L#10000;
      <D;
      );
      AN    DB7.DBX 130.1;
      AN    DB7.DBX 124.0;
      =     Q 1.3;
NETWORK
TITLE =
      A     M 10.0;
      =     L 0.0;
      A     L 0.0;
      A     T 48;
      =     Q 1.5;
      A     L 0.0;
      A     T 46;
      =     Q 1.4;
NETWORK
TITLE =
      O     M 52.1;
      O     M 31.7;
      O;
      A     T 43;
      AN    T 31;
      =     Q 1.6;
NETWORK
TITLE =
      A(;
      O     M 52.3;
      O     Q 1.7;
      O     M 32.0;
      );
      A     Q 0.3;
      A     M 10.0;
      =     Q 1.7;
NETWORK
TITLE =
      A     M 74.1;
      A     M 74.3;
      =     Q 32.2;
NETWORK
TITLE =
      O     M 74.2;
      O     M 74.4;
      =     Q 32.3;
NETWORK
TITLE =
      AN    M 10.0;
      =     Q 32.5;
NETWORK
TITLE =
      A(;
      O     M 11.2;
      O     M 11.4;
      );
      AN    M 30.1;
      AN    M 30.0;
      AN    Q 1.2;
      AN    Q 1.3;
      O;
      A     M 11.4;
      A     M 12.0;
      A     M 60.0;
      AN    M 50.0;
      AN    M 50.1;
      =     Q 32.6;
NETWORK
TITLE =
      A(;
      O     M 12.3;
      O     M 70.2;
      O     M 74.2;
      );
      A     M 1.1;
      =     L 0.0;
      A     L 0.0;
      AN    T 66;
      A     M 0.5;
      =     Q 32.7;
      A     L 0.0;
      BLD   102;
      L     S5T#20S;
      SD    T 66;
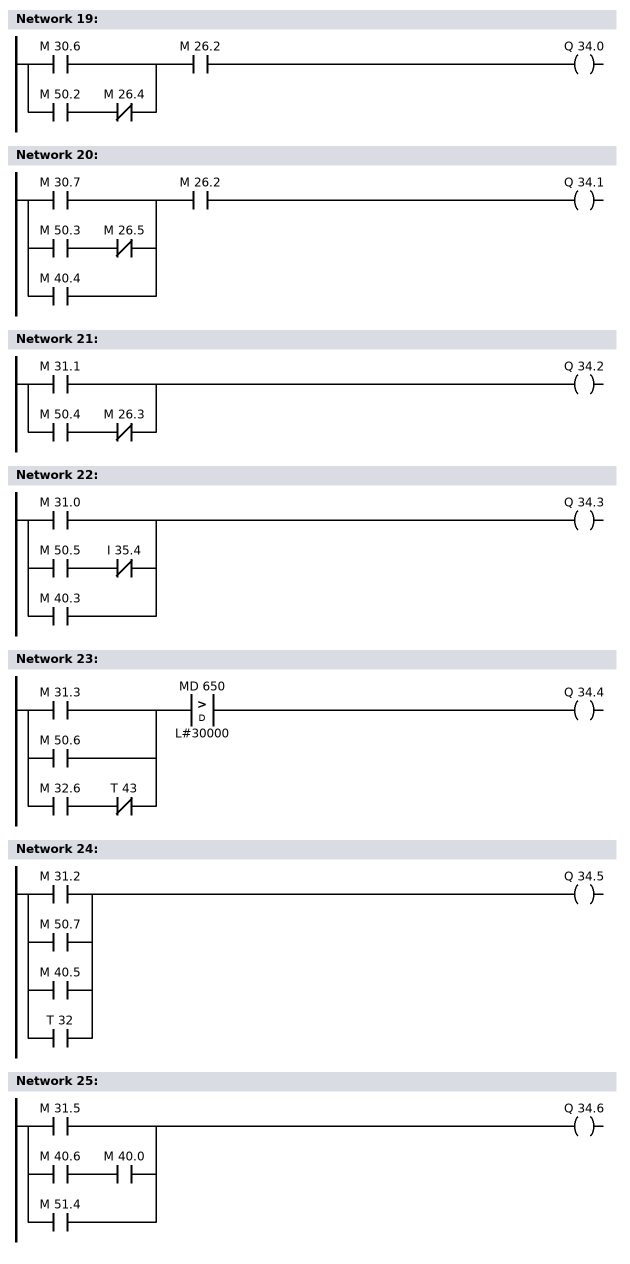
NETWORK
TITLE =
      A(;
      O     M 30.6;
      O;
      A     M 50.2;
      AN    M 26.4;
      );
      A     M 26.2;
      =     Q 34.0;
NETWORK
TITLE =
      A(;
      O     M 30.7;
      O;
      A     M 50.3;
      AN    M 26.5;
      O     M 40.4;
      );
      A     M 26.2;
      =     Q 34.1;
NETWORK
TITLE =
      O     M 31.1;
      O;
      A     M 50.4;
      AN    M 26.3;
      =     Q 34.2;
NETWORK
TITLE =
      O     M 31.0;
      O;
      A     M 50.5;
      AN    I 35.4;
      O     M 40.3;
      =     Q 34.3;
NETWORK
TITLE =
      A(;
      O     M 31.3;
      O     M 50.6;
      O;
      A     M 32.6;
      AN    T 43;
      );
      A(;
      L     MD 650;
      L     L#30000;
      >D;
      );
      =     Q 34.4;
NETWORK
TITLE =
      O     M 31.2;
      O     M 50.7;
      O     M 40.5;
      O     T 32;
      =     Q 34.5;
NETWORK
TITLE =
      O     M 31.5;
      O;
      A     M 40.6;
      A     M 40.0;
      O     M 51.4;
      =     Q 34.6;
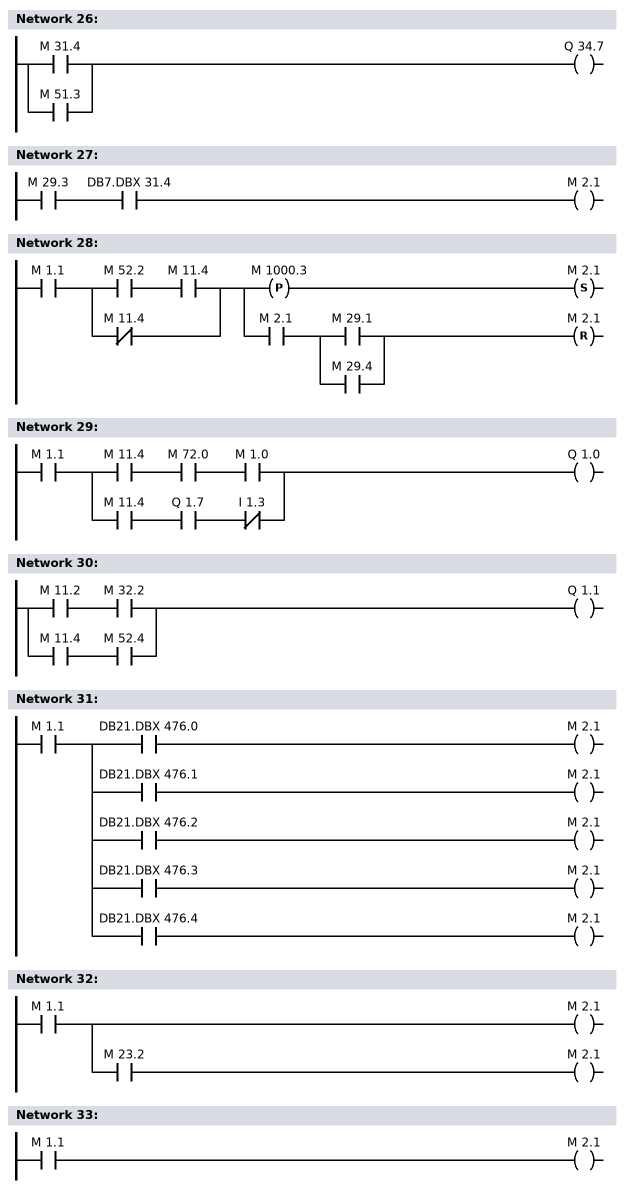
NETWORK
TITLE =
      O     M 31.4;
      O     M 51.3;
      =     Q 34.7;
NETWORK
TITLE =
      A     M 29.3;
      A     DB7.DBX 31.4;
      =     M 2.1;
NETWORK
TITLE =
      A     M 1.1;
      A(;
      A     M 52.2;
      A     M 11.4;
      ON    M 11.4;
      );
      =     L 0.0;
      A     L 0.0;
      FP    M 1000.3;
      S     M 2.1;
      A     L 0.0;
      A     M 2.1;
      A(;
      O     M 29.1;
      O     M 29.4;
      );
      R     M 2.1;
NETWORK
TITLE =
      A     M 1.1;
      A(;
      A     M 11.4;
      A     M 72.0;
      A     M 1.0;
      O;
      A     M 11.4;
      A     Q 1.7;
      AN    I 1.3;
      );
      =     Q 1.0;
NETWORK
TITLE =
      A     M 11.2;
      A     M 32.2;
      O;
      A     M 11.4;
      A     M 52.4;
      =     Q 1.1;
NETWORK
TITLE =
      A     M 1.1;
      =     L 0.0;
      A     L 0.0;
      A     DB21.DBX 476.0;
      =     M 2.1;
      A     L 0.0;
      A     DB21.DBX 476.1;
      =     M 2.1;
      A     L 0.0;
      A     DB21.DBX 476.2;
      =     M 2.1;
      A     L 0.0;
      A     DB21.DBX 476.3;
      =     M 2.1;
      A     L 0.0;
      A     DB21.DBX 476.4;
      =     M 2.1;
NETWORK
TITLE =
      A     M 1.1;
      =     L 0.0;
      A     L 0.0;
      BLD   102;
      =     M 2.1;
      A     L 0.0;
      A     M 23.2;
      =     M 2.1;
NETWORK
TITLE =
      A     M 1.1;
      =     M 2.1;
END_FUNCTION

FUNCTION FC 19 : VOID
VERSION : 0.1
BEGIN
// (block stored without names or comments; labels and parameter names are numbered)
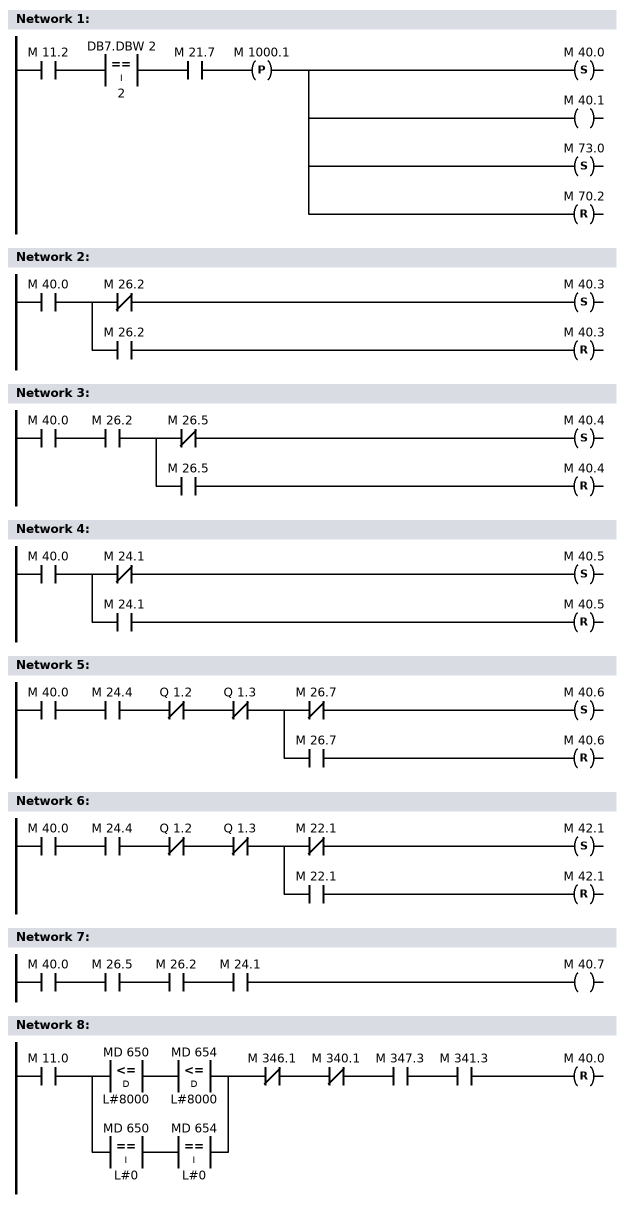
NETWORK
TITLE =
      A     M 11.2;
      A(;
      L     DB7.DBW 2;
      L     2;
      ==I;
      );
      A     M 21.7;
      FP    M 1000.1;
      S     M 40.0;
      =     M 40.1;
      S     M 73.0;
      R     M 70.2;
NETWORK
TITLE =
      A     M 40.0;
      =     L 0.0;
      A     L 0.0;
      AN    M 26.2;
      S     M 40.3;
      A     L 0.0;
      A     M 26.2;
      R     M 40.3;
NETWORK
TITLE =
      A     M 40.0;
      A     M 26.2;
      =     L 0.0;
      A     L 0.0;
      AN    M 26.5;
      S     M 40.4;
      A     L 0.0;
      A     M 26.5;
      R     M 40.4;
NETWORK
TITLE =
      A     M 40.0;
      =     L 0.0;
      A     L 0.0;
      AN    M 24.1;
      S     M 40.5;
      A     L 0.0;
      A     M 24.1;
      R     M 40.5;
NETWORK
TITLE =
      A     M 40.0;
      A     M 24.4;
      AN    Q 1.2;
      AN    Q 1.3;
      =     L 0.0;
      A     L 0.0;
      AN    M 26.7;
      S     M 40.6;
      A     L 0.0;
      A     M 26.7;
      R     M 40.6;
NETWORK
TITLE =
      A     M 40.0;
      A     M 24.4;
      AN    Q 1.2;
      AN    Q 1.3;
      =     L 0.0;
      A     L 0.0;
      AN    M 22.1;
      S     M 42.1;
      A     L 0.0;
      A     M 22.1;
      R     M 42.1;
NETWORK
TITLE =
      A     M 40.0;
      A     M 26.5;
      A     M 26.2;
      A     M 24.1;
      =     M 40.7;
NETWORK
TITLE =
      A     M 11.0;
      A(;
      A(;
      L     MD 650;
      L     L#8000;
      <=D;
      );
      A(;
      L     MD 654;
      L     L#8000;
      <=D;
      );
      O;
      A(;
      L     MD 650;
      L     L#0;
      ==I;
      );
      A(;
      L     MD 654;
      L     L#0;
      ==I;
      );
      );
      AN    M 346.1;
      AN    M 340.1;
      A     M 347.3;
      A     M 341.3;
      R     M 40.0;
NETWORK
TITLE =
END_FUNCTION

FUNCTION FC 24 : VOID
VERSION : 0.1
BEGIN
// (block stored without names or comments; labels and parameter names are numbered)
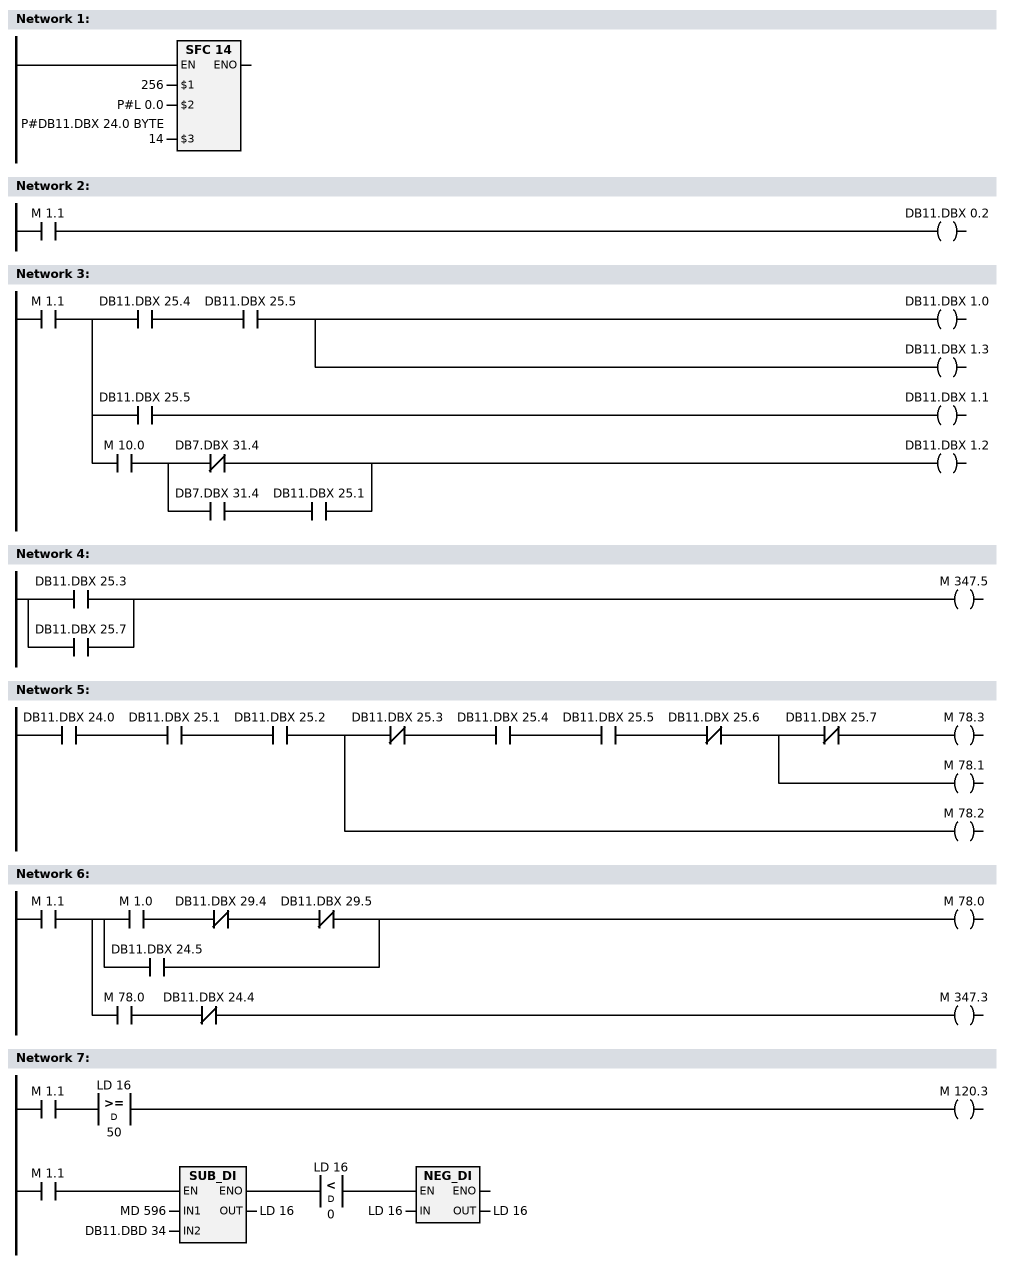
NETWORK
TITLE =
      CALL  SFC 14 (
           $1                       := 256,
           $2                       := P#L 0.0,
           $3                       := P#DB11.DBX 24.0 BYTE 14);
      NOP   0;
NETWORK
TITLE =
      A     M 1.1;
      =     DB11.DBX 0.2;
NETWORK
TITLE =
      A     M 1.1;
      =     L 21.0;
      A     L 21.0;
      A     DB11.DBX 25.4;
      A     DB11.DBX 25.5;
      =     DB11.DBX 1.0;
      =     DB11.DBX 1.3;
      A     L 21.0;
      A     DB11.DBX 25.5;
      =     DB11.DBX 1.1;
      A     L 21.0;
      A     M 10.0;
      A(;
      ON    DB7.DBX 31.4;
      O;
      A     DB7.DBX 31.4;
      A     DB11.DBX 25.1;
      );
      =     DB11.DBX 1.2;
NETWORK
TITLE =
      O     DB11.DBX 25.3;
      O     DB11.DBX 25.7;
      =     M 347.5;
NETWORK
TITLE =
      A     DB11.DBX 24.0;
      A     DB11.DBX 25.1;
      A     DB11.DBX 25.2;
      =     L 21.0;
      A     L 21.0;
      AN    DB11.DBX 25.3;
      A     DB11.DBX 25.4;
      A     DB11.DBX 25.5;
      AN    DB11.DBX 25.6;
      =     L 21.1;
      A     L 21.1;
      AN    DB11.DBX 25.7;
      =     M 78.3;
      A     L 21.1;
      BLD   102;
      =     M 78.1;
      A     L 21.0;
      BLD   102;
      =     M 78.2;
NETWORK
TITLE =
      A     M 1.1;
      =     L 21.0;
      A     L 21.0;
      A(;
      A     M 1.0;
      AN    DB11.DBX 29.4;
      AN    DB11.DBX 29.5;
      O     DB11.DBX 24.5;
      );
      =     M 78.0;
      A     L 21.0;
      A     M 78.0;
      AN    DB11.DBX 24.4;
      =     M 347.3;
NETWORK
TITLE =
      A     M 1.1;
      =     L 20.0;
      A(;
      A     L 20.0;
      JNB   M001;
      L     MD 596;
      L     DB11.DBD 34;
      -D;
      T     LD 16;
      AN    OV;
      SAVE;
      CLR;
M001: A     BR;
      );
      A(;
      L     LD 16;
      L     0;
      <D;
      );
      JNB   M002;
      L     LD 16;
      NEGD;
      T     LD 16;
M002: NOP   0;
      A     L 20.0;
      A(;
      L     LD 16;
      L     50;
      >=D;
      );
      =     M 120.3;
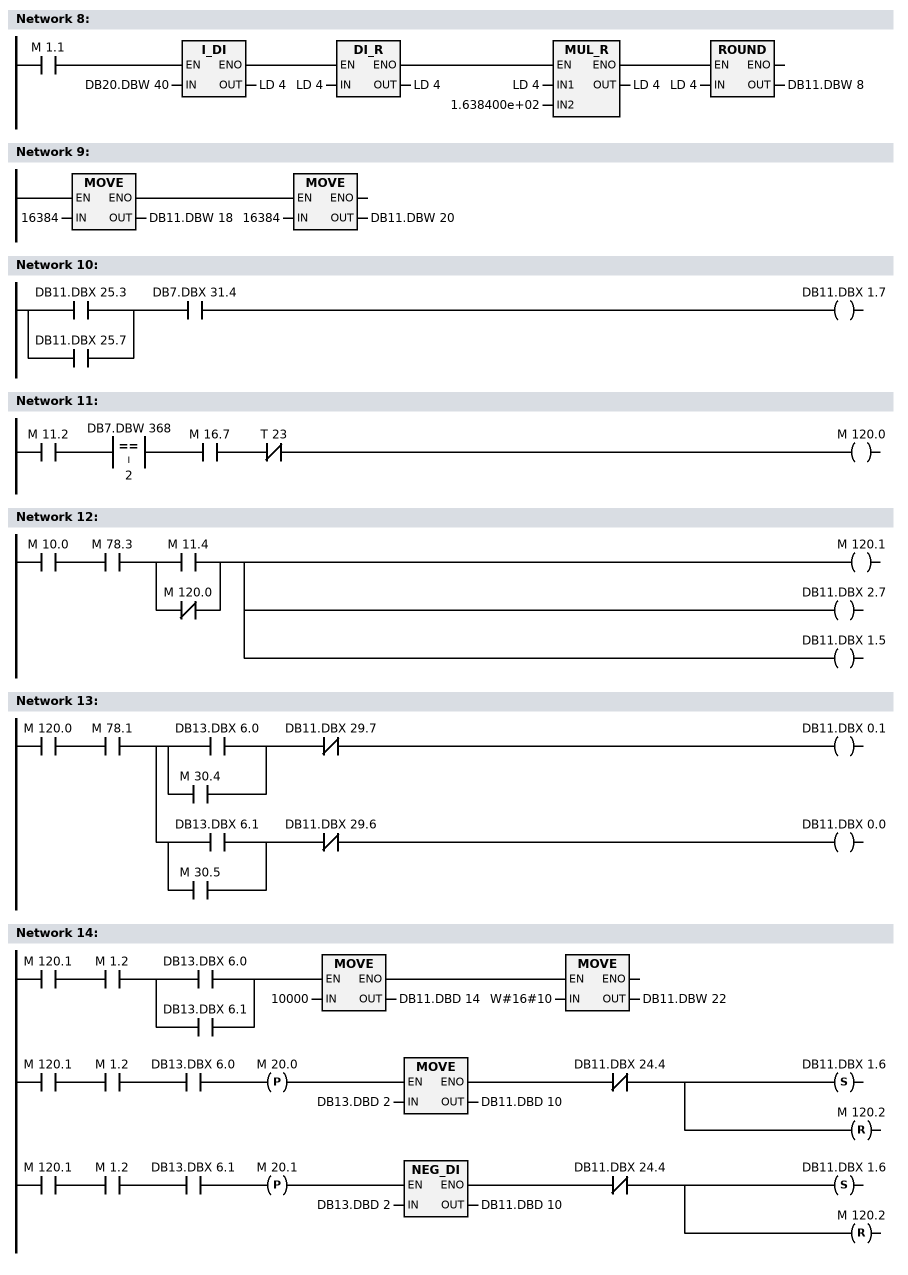
NETWORK
TITLE =
      A(;
      A(;
      A(;
      A     M 1.1;
      JNB   M003;
      L     DB20.DBW 40;
      ITD;
      T     LD 4;
      SET;
      SAVE;
      CLR;
M003: A     BR;
      );
      JNB   M004;
      L     LD 4;
      DTR;
      T     LD 4;
      SET;
      SAVE;
      CLR;
M004: A     BR;
      );
      JNB   M005;
      L     LD 4;
      L     1.638400e+02;
      *R;
      T     LD 4;
      AN    OV;
      SAVE;
      CLR;
M005: A     BR;
      );
      JNB   M006;
      L     LD 4;
      RND;
      T     DB11.DBW 8;
M006: NOP   0;
NETWORK
TITLE =
      A(;
      L     16384;
      T     DB11.DBW 18;
      SET;
      SAVE;
      CLR;
      A     BR;
      );
      JNB   M007;
      L     16384;
      T     DB11.DBW 20;
M007: NOP   0;
NETWORK
TITLE =
      A(;
      O     DB11.DBX 25.3;
      O     DB11.DBX 25.7;
      );
      A     DB7.DBX 31.4;
      =     DB11.DBX 1.7;
NETWORK
TITLE =
      A     M 11.2;
      A(;
      L     DB7.DBW 368;
      L     2;
      ==I;
      );
      A     M 16.7;
      AN    T 23;
      =     M 120.0;
NETWORK
TITLE =
      A     M 10.0;
      A     M 78.3;
      A(;
      O     M 11.4;
      ON    M 120.0;
      );
      =     M 120.1;
      =     DB11.DBX 2.7;
      =     DB11.DBX 1.5;
NETWORK
TITLE =
      A     M 120.0;
      A     M 78.1;
      =     L 21.0;
      A     L 21.0;
      A(;
      O     DB13.DBX 6.0;
      O     M 30.4;
      );
      AN    DB11.DBX 29.7;
      =     DB11.DBX 0.1;
      A     L 21.0;
      A(;
      O     DB13.DBX 6.1;
      O     M 30.5;
      );
      AN    DB11.DBX 29.6;
      =     DB11.DBX 0.0;
NETWORK
TITLE =
      A     M 120.1;
      A     M 1.2;
      =     L 21.0;
      A(;
      A     L 21.0;
      A(;
      O     DB13.DBX 6.0;
      O     DB13.DBX 6.1;
      );
      JNB   M008;
      L     10000;
      T     DB11.DBD 14;
      SET;
      SAVE;
      CLR;
M008: A     BR;
      );
      JNB   M009;
      L     W#16#10;
      T     DB11.DBW 22;
M009: NOP   0;
      A(;
      A     L 21.0;
      A     DB13.DBX 6.0;
      FP    M 20.0;
      JNB   M010;
      L     DB13.DBD 2;
      T     DB11.DBD 10;
      SET;
      SAVE;
      CLR;
M010: A     BR;
      );
      AN    DB11.DBX 24.4;
      S     DB11.DBX 1.6;
      R     M 120.2;
      A(;
      A     L 21.0;
      A     DB13.DBX 6.1;
      FP    M 20.1;
      JNB   M011;
      L     DB13.DBD 2;
      NEGD;
      T     DB11.DBD 10;
      AN    OV;
      SAVE;
      CLR;
M011: A     BR;
      );
      AN    DB11.DBX 24.4;
      S     DB11.DBX 1.6;
      R     M 120.2;
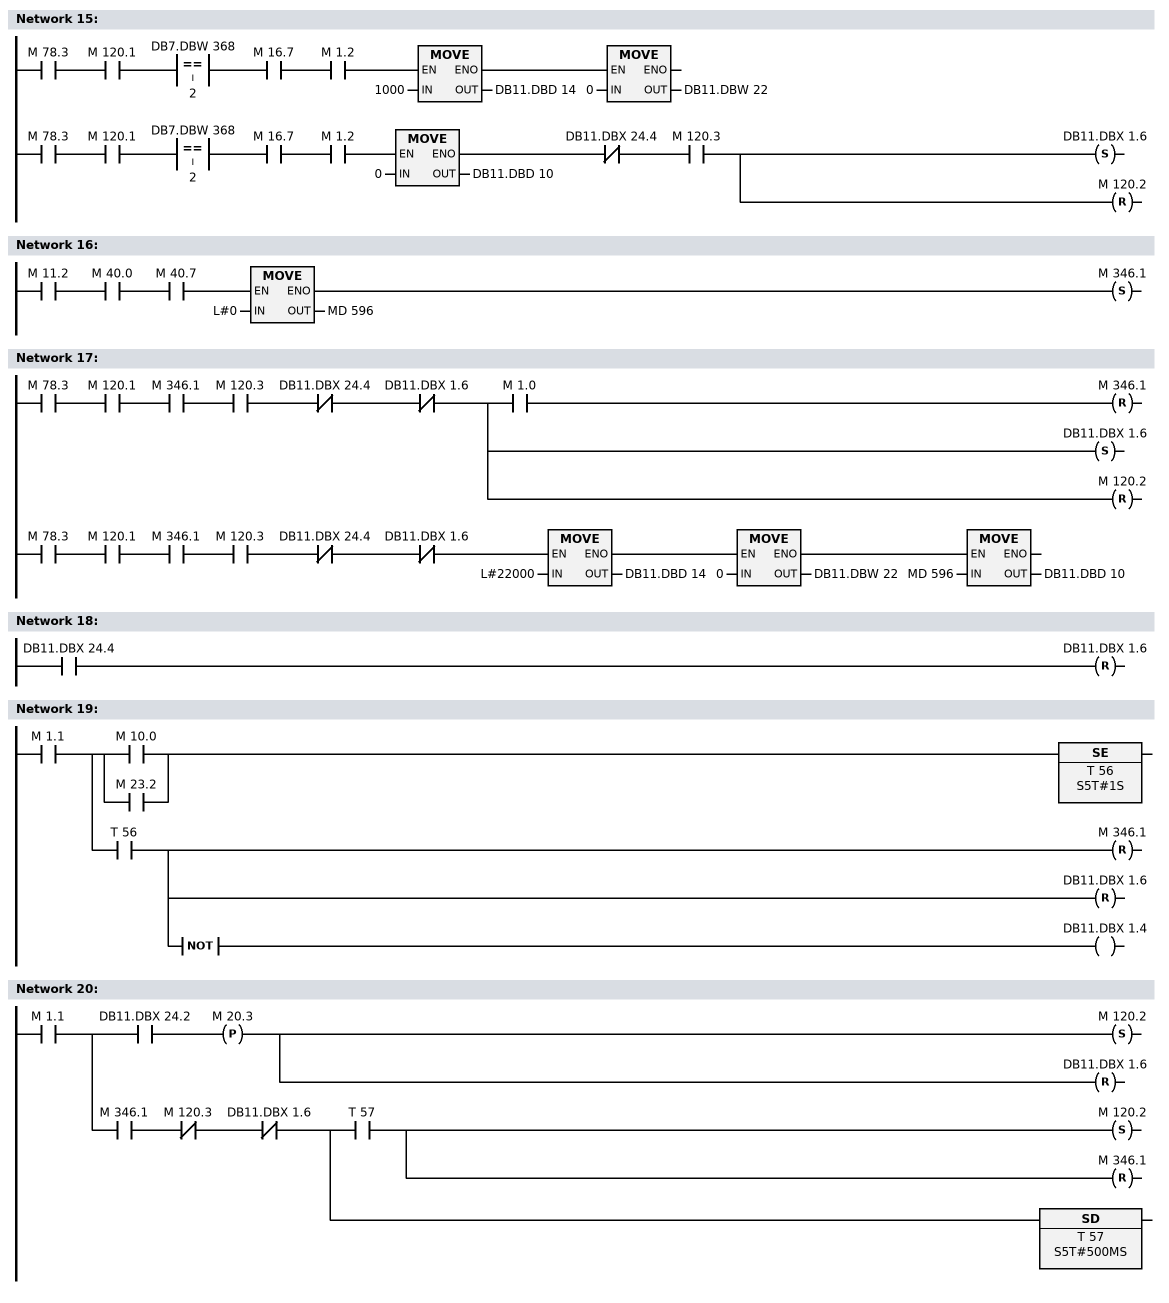
NETWORK
TITLE =
      A     M 78.3;
      A     M 120.1;
      A(;
      L     DB7.DBW 368;
      L     2;
      ==I;
      );
      A     M 16.7;
      =     L 21.0;
      A(;
      A     L 21.0;
      A     M 1.2;
      JNB   M012;
      L     1000;
      T     DB11.DBD 14;
      SET;
      SAVE;
      CLR;
M012: A     BR;
      );
      JNB   M013;
      L     0;
      T     DB11.DBW 22;
M013: NOP   0;
      A(;
      A     L 21.0;
      A     M 1.2;
      JNB   M014;
      L     0;
      T     DB11.DBD 10;
      SET;
      SAVE;
      CLR;
M014: A     BR;
      );
      AN    DB11.DBX 24.4;
      A     M 120.3;
      S     DB11.DBX 1.6;
      R     M 120.2;
NETWORK
TITLE =
      A     M 11.2;
      A     M 40.0;
      A     M 40.7;
      JNB   M015;
      L     L#0;
      T     MD 596;
      SET;
      SAVE;
      CLR;
M015: A     BR;
      S     M 346.1;
NETWORK
TITLE =
      A     M 78.3;
      A     M 120.1;
      A     M 346.1;
      A     M 120.3;
      AN    DB11.DBX 24.4;
      AN    DB11.DBX 1.6;
      =     L 21.0;
      A(;
      A(;
      A     L 21.0;
      JNB   M016;
      L     L#22000;
      T     DB11.DBD 14;
      SET;
      SAVE;
      CLR;
M016: A     BR;
      );
      JNB   M017;
      L     0;
      T     DB11.DBW 22;
      SET;
      SAVE;
      CLR;
M017: A     BR;
      );
      JNB   M018;
      L     MD 596;
      T     DB11.DBD 10;
M018: NOP   0;
      A     L 21.0;
      A     M 1.0;
      R     M 346.1;
      A     L 21.0;
      BLD   102;
      S     DB11.DBX 1.6;
      A     L 21.0;
      BLD   102;
      R     M 120.2;
NETWORK
TITLE =
      A     DB11.DBX 24.4;
      R     DB11.DBX 1.6;
NETWORK
TITLE =
      A     M 1.1;
      =     L 21.0;
      A     L 21.0;
      A(;
      O     M 10.0;
      O     M 23.2;
      );
      L     S5T#1S;
      SE    T 56;
      A     L 21.0;
      A     T 56;
      =     L 21.1;
      A     L 21.1;
      BLD   102;
      R     M 346.1;
      A     L 21.1;
      BLD   102;
      R     DB11.DBX 1.6;
      A     L 21.1;
      NOT;
      =     DB11.DBX 1.4;
NETWORK
TITLE =
      A     M 1.1;
      =     L 21.0;
      A     L 21.0;
      A     DB11.DBX 24.2;
      FP    M 20.3;
      S     M 120.2;
      R     DB11.DBX 1.6;
      A     L 21.0;
      A     M 346.1;
      AN    M 120.3;
      AN    DB11.DBX 1.6;
      =     L 21.1;
      A     L 21.1;
      A     T 57;
      S     M 120.2;
      R     M 346.1;
      A     L 21.1;
      BLD   102;
      L     S5T#500MS;
      SD    T 57;
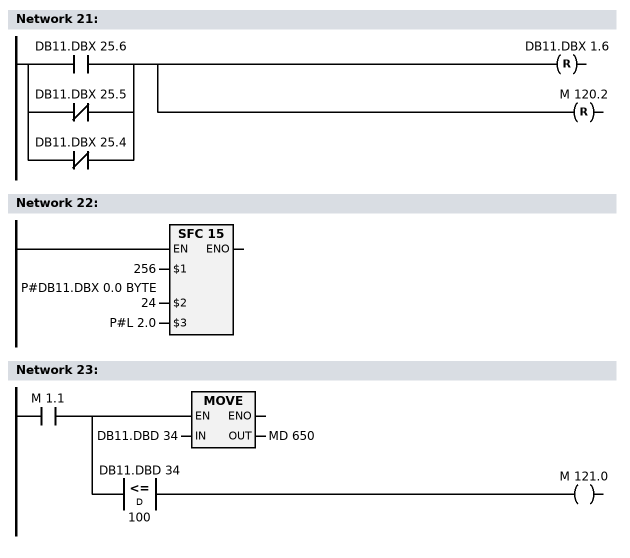
NETWORK
TITLE =
      O     DB11.DBX 25.6;
      ON    DB11.DBX 25.5;
      ON    DB11.DBX 25.4;
      R     DB11.DBX 1.6;
      R     M 120.2;
NETWORK
TITLE =
      CALL  SFC 15 (
           $1                       := 256,
           $2                       := P#DB11.DBX 0.0 BYTE 24,
           $3                       := P#L 2.0);
      NOP   0;
NETWORK
TITLE =
      A     M 1.1;
      =     L 20.0;
      A     L 20.0;
      JNB   M019;
      L     DB11.DBD 34;
      T     MD 650;
M019: NOP   0;
      A     L 20.0;
      A(;
      L     DB11.DBD 34;
      L     100;
      <=D;
      );
      =     M 121.0;
END_FUNCTION

FUNCTION FC 25 : VOID
VERSION : 0.1
BEGIN
// (block stored without names or comments; labels and parameter names are numbered)
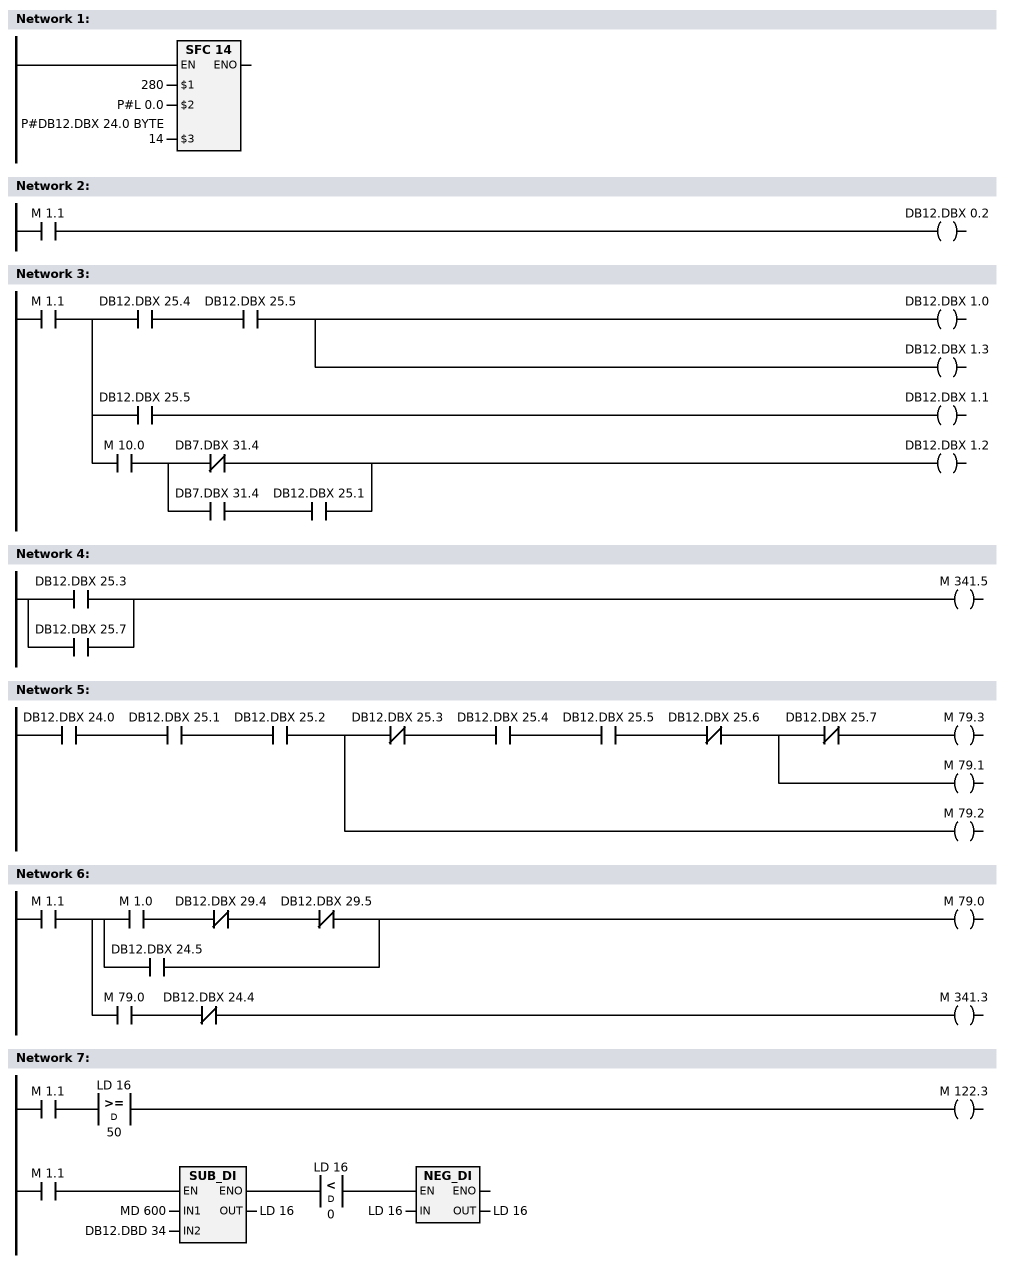
NETWORK
TITLE =
      CALL  SFC 14 (
           $1                       := 280,
           $2                       := P#L 0.0,
           $3                       := P#DB12.DBX 24.0 BYTE 14);
      NOP   0;
NETWORK
TITLE =
      A     M 1.1;
      =     DB12.DBX 0.2;
NETWORK
TITLE =
      A     M 1.1;
      =     L 21.0;
      A     L 21.0;
      A     DB12.DBX 25.4;
      A     DB12.DBX 25.5;
      =     DB12.DBX 1.0;
      =     DB12.DBX 1.3;
      A     L 21.0;
      A     DB12.DBX 25.5;
      =     DB12.DBX 1.1;
      A     L 21.0;
      A     M 10.0;
      A(;
      ON    DB7.DBX 31.4;
      O;
      A     DB7.DBX 31.4;
      A     DB12.DBX 25.1;
      );
      =     DB12.DBX 1.2;
NETWORK
TITLE =
      O     DB12.DBX 25.3;
      O     DB12.DBX 25.7;
      =     M 341.5;
NETWORK
TITLE =
      A     DB12.DBX 24.0;
      A     DB12.DBX 25.1;
      A     DB12.DBX 25.2;
      =     L 21.0;
      A     L 21.0;
      AN    DB12.DBX 25.3;
      A     DB12.DBX 25.4;
      A     DB12.DBX 25.5;
      AN    DB12.DBX 25.6;
      =     L 21.1;
      A     L 21.1;
      AN    DB12.DBX 25.7;
      =     M 79.3;
      A     L 21.1;
      BLD   102;
      =     M 79.1;
      A     L 21.0;
      BLD   102;
      =     M 79.2;
NETWORK
TITLE =
      A     M 1.1;
      =     L 21.0;
      A     L 21.0;
      A(;
      A     M 1.0;
      AN    DB12.DBX 29.4;
      AN    DB12.DBX 29.5;
      O     DB12.DBX 24.5;
      );
      =     M 79.0;
      A     L 21.0;
      A     M 79.0;
      AN    DB12.DBX 24.4;
      =     M 341.3;
NETWORK
TITLE =
      A     M 1.1;
      =     L 20.0;
      A(;
      A     L 20.0;
      JNB   M001;
      L     MD 600;
      L     DB12.DBD 34;
      -D;
      T     LD 16;
      AN    OV;
      SAVE;
      CLR;
M001: A     BR;
      );
      A(;
      L     LD 16;
      L     0;
      <D;
      );
      JNB   M002;
      L     LD 16;
      NEGD;
      T     LD 16;
M002: NOP   0;
      A     L 20.0;
      A(;
      L     LD 16;
      L     50;
      >=D;
      );
      =     M 122.3;
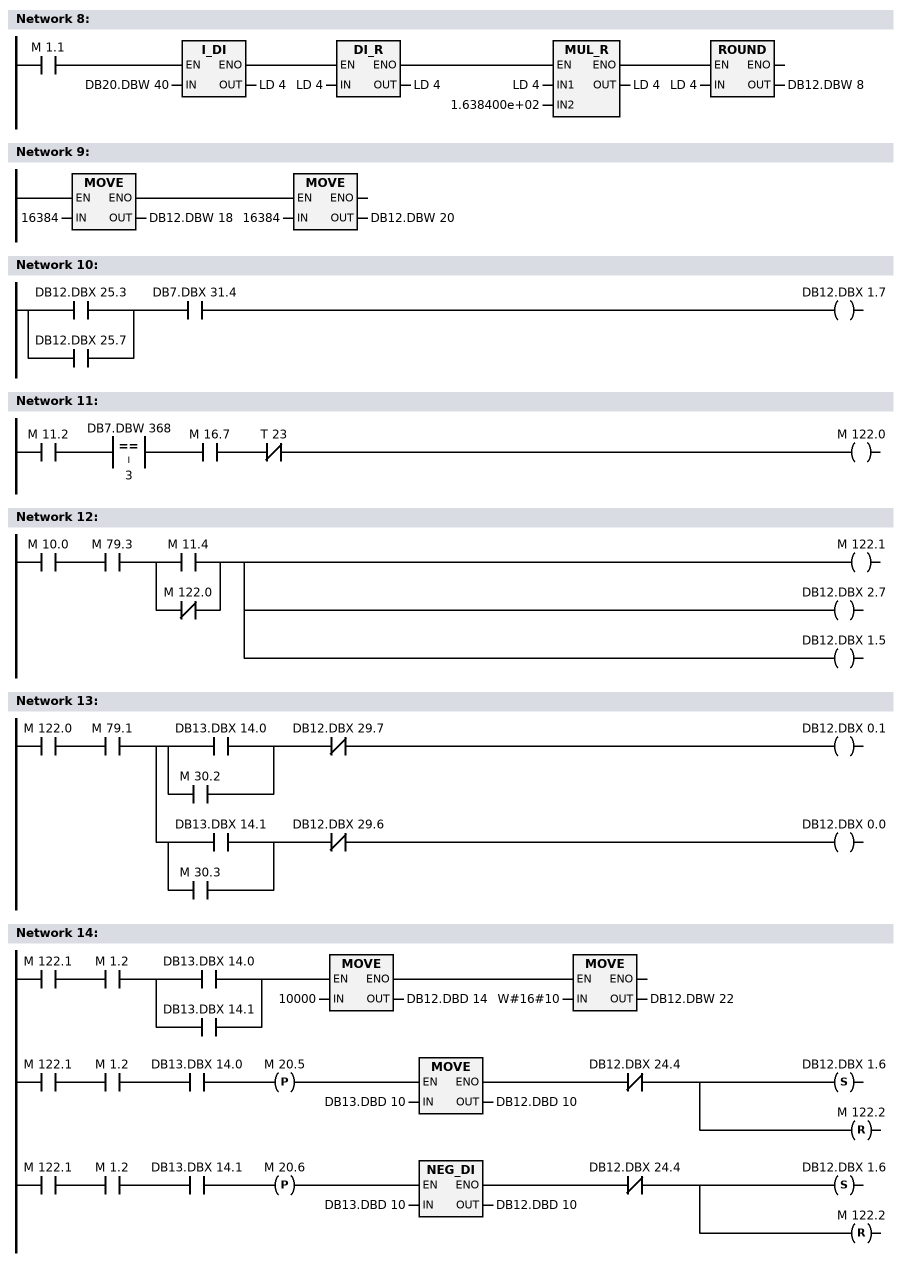
NETWORK
TITLE =
      A(;
      A(;
      A(;
      A     M 1.1;
      JNB   M003;
      L     DB20.DBW 40;
      ITD;
      T     LD 4;
      SET;
      SAVE;
      CLR;
M003: A     BR;
      );
      JNB   M004;
      L     LD 4;
      DTR;
      T     LD 4;
      SET;
      SAVE;
      CLR;
M004: A     BR;
      );
      JNB   M005;
      L     LD 4;
      L     1.638400e+02;
      *R;
      T     LD 4;
      AN    OV;
      SAVE;
      CLR;
M005: A     BR;
      );
      JNB   M006;
      L     LD 4;
      RND;
      T     DB12.DBW 8;
M006: NOP   0;
NETWORK
TITLE =
      A(;
      L     16384;
      T     DB12.DBW 18;
      SET;
      SAVE;
      CLR;
      A     BR;
      );
      JNB   M007;
      L     16384;
      T     DB12.DBW 20;
M007: NOP   0;
NETWORK
TITLE =
      A(;
      O     DB12.DBX 25.3;
      O     DB12.DBX 25.7;
      );
      A     DB7.DBX 31.4;
      =     DB12.DBX 1.7;
NETWORK
TITLE =
      A     M 11.2;
      A(;
      L     DB7.DBW 368;
      L     3;
      ==I;
      );
      A     M 16.7;
      AN    T 23;
      =     M 122.0;
NETWORK
TITLE =
      A     M 10.0;
      A     M 79.3;
      A(;
      O     M 11.4;
      ON    M 122.0;
      );
      =     M 122.1;
      =     DB12.DBX 2.7;
      =     DB12.DBX 1.5;
NETWORK
TITLE =
      A     M 122.0;
      A     M 79.1;
      =     L 21.0;
      A     L 21.0;
      A(;
      O     DB13.DBX 14.0;
      O     M 30.2;
      );
      AN    DB12.DBX 29.7;
      =     DB12.DBX 0.1;
      A     L 21.0;
      A(;
      O     DB13.DBX 14.1;
      O     M 30.3;
      );
      AN    DB12.DBX 29.6;
      =     DB12.DBX 0.0;
NETWORK
TITLE =
      A     M 122.1;
      A     M 1.2;
      =     L 21.0;
      A(;
      A     L 21.0;
      A(;
      O     DB13.DBX 14.0;
      O     DB13.DBX 14.1;
      );
      JNB   M008;
      L     10000;
      T     DB12.DBD 14;
      SET;
      SAVE;
      CLR;
M008: A     BR;
      );
      JNB   M009;
      L     W#16#10;
      T     DB12.DBW 22;
M009: NOP   0;
      A(;
      A     L 21.0;
      A     DB13.DBX 14.0;
      FP    M 20.5;
      JNB   M010;
      L     DB13.DBD 10;
      T     DB12.DBD 10;
      SET;
      SAVE;
      CLR;
M010: A     BR;
      );
      AN    DB12.DBX 24.4;
      S     DB12.DBX 1.6;
      R     M 122.2;
      A(;
      A     L 21.0;
      A     DB13.DBX 14.1;
      FP    M 20.6;
      JNB   M011;
      L     DB13.DBD 10;
      NEGD;
      T     DB12.DBD 10;
      AN    OV;
      SAVE;
      CLR;
M011: A     BR;
      );
      AN    DB12.DBX 24.4;
      S     DB12.DBX 1.6;
      R     M 122.2;
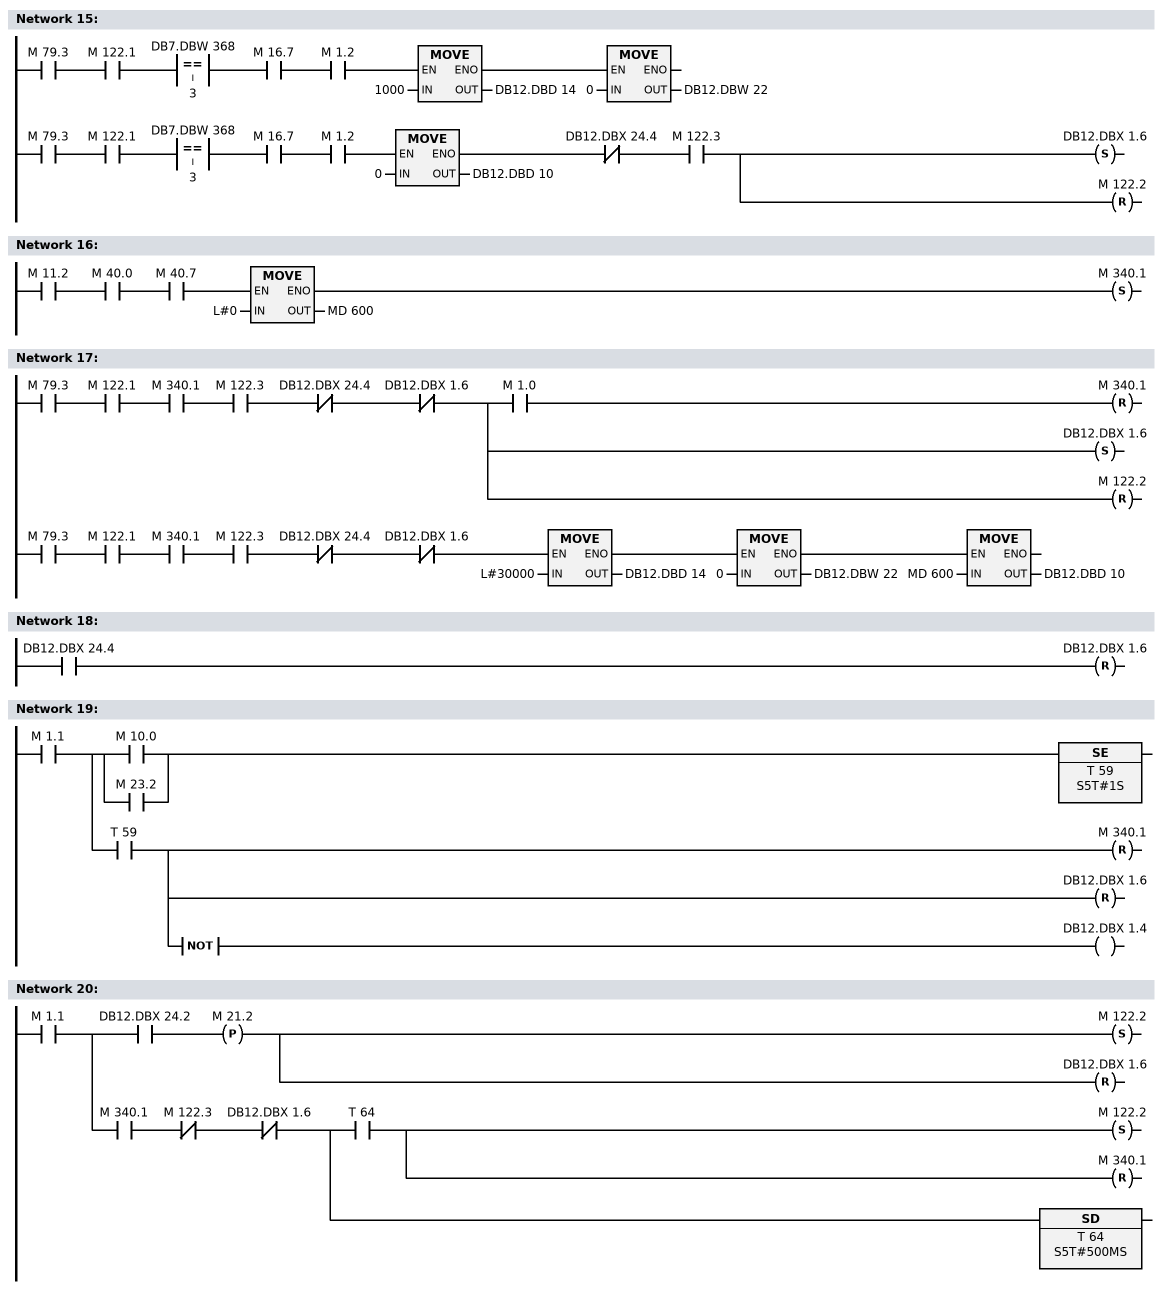
NETWORK
TITLE =
      A     M 79.3;
      A     M 122.1;
      A(;
      L     DB7.DBW 368;
      L     3;
      ==I;
      );
      A     M 16.7;
      =     L 21.0;
      A(;
      A     L 21.0;
      A     M 1.2;
      JNB   M012;
      L     1000;
      T     DB12.DBD 14;
      SET;
      SAVE;
      CLR;
M012: A     BR;
      );
      JNB   M013;
      L     0;
      T     DB12.DBW 22;
M013: NOP   0;
      A(;
      A     L 21.0;
      A     M 1.2;
      JNB   M014;
      L     0;
      T     DB12.DBD 10;
      SET;
      SAVE;
      CLR;
M014: A     BR;
      );
      AN    DB12.DBX 24.4;
      A     M 122.3;
      S     DB12.DBX 1.6;
      R     M 122.2;
NETWORK
TITLE =
      A     M 11.2;
      A     M 40.0;
      A     M 40.7;
      JNB   M015;
      L     L#0;
      T     MD 600;
      SET;
      SAVE;
      CLR;
M015: A     BR;
      S     M 340.1;
NETWORK
TITLE =
      A     M 79.3;
      A     M 122.1;
      A     M 340.1;
      A     M 122.3;
      AN    DB12.DBX 24.4;
      AN    DB12.DBX 1.6;
      =     L 21.0;
      A(;
      A(;
      A     L 21.0;
      JNB   M016;
      L     L#30000;
      T     DB12.DBD 14;
      SET;
      SAVE;
      CLR;
M016: A     BR;
      );
      JNB   M017;
      L     0;
      T     DB12.DBW 22;
      SET;
      SAVE;
      CLR;
M017: A     BR;
      );
      JNB   M018;
      L     MD 600;
      T     DB12.DBD 10;
M018: NOP   0;
      A     L 21.0;
      A     M 1.0;
      R     M 340.1;
      A     L 21.0;
      BLD   102;
      S     DB12.DBX 1.6;
      A     L 21.0;
      BLD   102;
      R     M 122.2;
NETWORK
TITLE =
      A     DB12.DBX 24.4;
      R     DB12.DBX 1.6;
NETWORK
TITLE =
      A     M 1.1;
      =     L 21.0;
      A     L 21.0;
      A(;
      O     M 10.0;
      O     M 23.2;
      );
      L     S5T#1S;
      SE    T 59;
      A     L 21.0;
      A     T 59;
      =     L 21.1;
      A     L 21.1;
      BLD   102;
      R     M 340.1;
      A     L 21.1;
      BLD   102;
      R     DB12.DBX 1.6;
      A     L 21.1;
      NOT;
      =     DB12.DBX 1.4;
NETWORK
TITLE =
      A     M 1.1;
      =     L 21.0;
      A     L 21.0;
      A     DB12.DBX 24.2;
      FP    M 21.2;
      S     M 122.2;
      R     DB12.DBX 1.6;
      A     L 21.0;
      A     M 340.1;
      AN    M 122.3;
      AN    DB12.DBX 1.6;
      =     L 21.1;
      A     L 21.1;
      A     T 64;
      S     M 122.2;
      R     M 340.1;
      A     L 21.1;
      BLD   102;
      L     S5T#500MS;
      SD    T 64;
